LIN {X 0,Y 433.901,Z 245.879,A -85,B 0,C 180,E1 -10138.023,E2 -10138.023} C_VEL
LIN {X 0,Y 437.066,Z 265.172,A -85,B 0,C 180,E1 -10138.671,E2 -10138.671} C_VEL
LIN {X 0,Y 434.096,Z 394.919,A -85,B 0,C 180,E1 -10140.942,E2 -10140.942} C_VEL
LIN {X 0,Y 433.119,Z 438.839,A -85,B 0,C 180,E1 -10141.742,E2 -10141.742} C_VEL
LIN {X 0,Y 432.141,Z 454.828,A -85,B 0,C 180,E1 -10142.19,E2 -10142.19} C_VEL
LIN {X 0,Y 431.054,Z 471,A -85,B 0,C 180,E1 -10142.838,E2 -10142.838} C_VEL
LIN {X 0,Y 429.617,Z 486.877,A -85,B 0,C 180,E1 -10143.658,E2 -10143.658} C_VEL
LIN {X 0,Y 428.212,Z 501.806,A -85,B 0,C 180,E1 -10144.632,E2 -10144.632} C_VEL
LIN {X 0,Y 426.513,Z 516.607,A -85,B 0,C 180,E1 -10145.803,E2 -10145.803} C_VEL
LIN {X 0,Y 424.863,Z 530.394,A -85,B 0,C 180,E1 -10147.125,E2 -10147.125} C_VEL
LIN {X 0,Y 423.301,Z 543.183,A -85,B 0,C 180,E1 -10148.577,E2 -10148.577} C_VEL
LIN {X 0,Y 421.945,Z 554.232,A -85,B 0,C 180,E1 -10150.035,E2 -10150.035} C_VEL
LIN {X 0,Y 420.588,Z 565.241,A -85,B 0,C 180,E1 -10151.742,E2 -10151.742} C_VEL
LIN {X 0,Y 419.49,Z 575.91,A -85,B 0,C 180,E1 -10153.703,E2 -10153.703} C_VEL
LIN {X 0,Y 418.494,Z 584.872,A -85,B 0,C 180,E1 -10155.659,E2 -10155.659} C_VEL
LIN {X 0,Y 417.936,Z 591.553,A -85,B 0,C 180,E1 -10157.373,E2 -10157.373} C_VEL
LIN {X 0,Y 417.496,Z 597.846,A -85,B 0,C 180,E1 -10159.329,E2 -10159.329} C_VEL
LIN {X 0,Y 417.2,Z 603.006,A -85,B 0,C 180,E1 -10161.28,E2 -10161.28} C_VEL
LIN {X 0,Y 417.134,Z 607.023,A -85,B 0,C 180,E1 -10163.227,E2 -10163.227} C_VEL
LIN {X 0,Y 417.018,Z 609.993,A -85,B 0,C 180,E1 -10165.167,E2 -10165.167} C_VEL
LIN {X 0,Y 417.006,Z 611.955,A -85,B 0,C 180,E1 -10167.102,E2 -10167.102} C_VEL
LIN {X 0,Y 417.009,Z 612.924,A -85,B 0,C 180,E1 -10169.035,E2 -10169.035} C_VEL
LIN {X 0,Y 417.009,Z 612.93,A -85,B 0,C 180,E1 -10170.966,E2 -10170.966} C_VEL
LIN {X 0,Y 417.006,Z 611.951,A -85,B 0,C 180,E1 -10172.898,E2 -10172.898} C_VEL
LIN {X 0,Y 417.019,Z 609.997,A -85,B 0,C 180,E1 -10174.834,E2 -10174.834} C_VEL
LIN {X 0,Y 417.134,Z 607.013,A -85,B 0,C 180,E1 -10176.773,E2 -10176.773} C_VEL
LIN {X 0,Y 417.202,Z 602.998,A -85,B 0,C 180,E1 -10178.72,E2 -10178.72} C_VEL
LIN {X 0,Y 417.496,Z 597.807,A -85,B 0,C 180,E1 -10180.671,E2 -10180.671} C_VEL
LIN {X 0,Y 418.041,Z 590.748,A -85,B 0,C 180,E1 -10182.819,E2 -10182.819} C_VEL
LIN {X 0,Y 418.673,Z 582.701,A -85,B 0,C 180,E1 -10184.832,E2 -10184.832} C_VEL
LIN {X 0,Y 419.692,Z 573.308,A -85,B 0,C 180,E1 -10186.776,E2 -10186.776} C_VEL
LIN {X 0,Y 420.73,Z 563.461,A -85,B 0,C 180,E1 -10188.505,E2 -10188.505} C_VEL
LIN {X 0,Y 422.098,Z 552.064,A -85,B 0,C 180,E1 -10190.212,E2 -10190.212} C_VEL
LIN {X 0,Y 423.494,Z 540.698,A -85,B 0,C 180,E1 -10191.669,E2 -10191.669} C_VEL
LIN {X 0,Y 425.098,Z 527.299,A -85,B 0,C 180,E1 -10193.12,E2 -10193.12} C_VEL
LIN {X 0,Y 426.529,Z 514.146,A -85,B 0,C 180,E1 -10194.326,E2 -10194.326} C_VEL
LIN {X 0,Y 428.112,Z 499.325,A -85,B 0,C 180,E1 -10195.459,E2 -10195.459} C_VEL
LIN {X 0,Y 429.661,Z 484.109,A -85,B 0,C 180,E1 -10196.405,E2 -10196.405} C_VEL
LIN {X 0,Y 430.887,Z 468.48,A -85,B 0,C 180,E1 -10197.174,E2 -10197.174} C_VEL
LIN {X 0,Y 431.837,Z 452.772,A -85,B 0,C 180,E1 -10197.766,E2 -10197.766} C_VEL
LIN {X 0,Y 432.796,Z 435.249,A -85,B 0,C 180,E1 -10198.212,E2 -10198.212} C_VEL
LIN {X 0,Y 436.415,Z 265.637,A -85,B 0,C 180,E1 -10201.169,E2 -10201.169} C_VEL
LIN {X 0,Y 432.886,Z 244.933,A -85,B 0,C 180,E1 -10201.842,E2 -10201.842} C_VEL
LIN {X 0,Y 426.31,Z 230.903,A -85,B 0,C 180,E1 -10202.655,E2 -10202.655} C_VEL
LIN {X 0,Y 421.236,Z 214.637,A -85,B 0,C 180,E1 -10205.162,E2 -10205.162} C_VEL
LIN {X 0,Y 418.237,Z 205.705,A -85,B 0,C 180,E1 -10206.62,E2 -10206.62} C_VEL
LIN {X 0,Y 418.241,Z 205.695,A -85,B 0,C 180,E1 -10209.683,E2 -10209.683} C_VEL
LIN {X 0,Y 418.221,Z 205.698,A -85,B 0,C 180,E1 -10212.32,E2 -10212.32} C_VEL
LIN {X 0,Y 418.233,Z 205.696,A -85,B 0,C 180,E1 -10215.109,E2 -10215.109} C_VEL
LIN {X 0,Y 418.231,Z 205.701,A -85,B 0,C 180,E1 -10217.766,E2 -10217.766} C_VEL
LIN {X 0,Y 418.242,Z 205.7,A -85,B 0,C 180,E1 -10221.557,E2 -10221.557} C_VEL
LIN {X 0,Y 418.255,Z 205.699,A -85,B 0,C 180,E1 -10225.159,E2 -10225.159} C_VEL
LIN {X 0,Y 418.242,Z 205.69,A -85,B 0,C 180,E1 -10227.472,E2 -10227.472} C_VEL
LIN {X 0,Y 418.266,Z 205.7,A -85,B 0,C 180,E1 -10230.895,E2 -10230.895} C_VEL
LIN {X 0,Y 418.265,Z 205.679,A -85,B 0,C 180,E1 -10234.096,E2 -10234.096} C_VEL
LIN {X 0,Y 418.235,Z 205.7,A -85,B 0,C 180,E1 -10237.264,E2 -10237.264} C_VEL
LIN {X 0,Y 418.28,Z 205.676,A -85,B 0,C 180,E1 -10240.364,E2 -10240.364} C_VEL
LIN {X 0,Y 418.313,Z 205.687,A -85,B 0,C 180,E1 -10243.405,E2 -10243.405} C_VEL
LIN {X 0,Y 418.343,Z 205.669,A -85,B 0,C 180,E1 -10246.999,E2 -10246.999} C_VEL
LIN {X 0,Y 418.336,Z 205.676,A -85,B 0,C 180,E1 -10250.329,E2 -10250.329} C_VEL
LIN {X 0,Y 418.468,Z 205.668,A -85,B 0,C 180,E1 -10253.249,E2 -10253.249} C_VEL
LIN {X 0,Y 418.332,Z 205.673,A -85,B 0,C 180,E1 -10255.181,E2 -10255.181} C_VEL
LIN {X 0,Y 418.539,Z 205.636,A -85,B 0,C 180,E1 -10258.075,E2 -10258.075} C_VEL
LIN {X 0,Y 418.667,Z 205.639,A -85,B 0,C 180,E1 -10260,E2 -10260} C_VEL
LIN {X 0,Y 418.497,Z 205.662,A -85,B 0,C 180,E1 -10262.888,E2 -10262.888} C_VEL
LIN {X 0,Y 418.49,Z 205.664,A -85,B 0,C 180,E1 -10266.751,E2 -10266.751} C_VEL
LIN {X 0,Y 418.337,Z 205.686,A -85,B 0,C 180,E1 -10269.671,E2 -10269.671} C_VEL
LIN {X 0,Y 418.344,Z 205.675,A -85,B 0,C 180,E1 -10273.001,E2 -10273.001} C_VEL
LIN {X 0,Y 418.31,Z 205.684,A -85,B 0,C 180,E1 -10276.736,E2 -10276.736} C_VEL
LIN {X 0,Y 418.268,Z 205.683,A -85,B 0,C 180,E1 -10279.79,E2 -10279.79} C_VEL
LIN {X 0,Y 418.236,Z 205.696,A -85,B 0,C 180,E1 -10282.736,E2 -10282.736} C_VEL
LIN {X 0,Y 418.268,Z 205.683,A -85,B 0,C 180,E1 -10285.904,E2 -10285.904} C_VEL
LIN {X 0,Y 418.272,Z 205.694,A -85,B 0,C 180,E1 -10289.161,E2 -10289.161} C_VEL
LIN {X 0,Y 418.255,Z 205.686,A -85,B 0,C 180,E1 -10292.844,E2 -10292.844} C_VEL
LIN {X 0,Y 418.246,Z 205.694,A -85,B 0,C 180,E1 -10296.239,E2 -10296.239} C_VEL
LIN {X 0,Y 418.253,Z 205.695,A -85,B 0,C 180,E1 -10299.682,E2 -10299.682} C_VEL
LIN {X 0,Y 418.227,Z 205.696,A -85,B 0,C 180,E1 -10302.321,E2 -10302.321} C_VEL
LIN {X 0,Y 418.234,Z 205.694,A -85,B 0,C 180,E1 -10305.109,E2 -10305.109} C_VEL
LIN {X 0,Y 418.238,Z 205.695,A -85,B 0,C 180,E1 -10307.767,E2 -10307.767} C_VEL
LIN {X 0,Y 418.243,Z 205.695,A -85,B 0,C 180,E1 -10310.621,E2 -10310.621} C_VEL
LIN {X 0,Y 418.241,Z 205.689,A -85,B 0,C 180,E1 -10313.976,E2 -10313.976} C_VEL
LIN {X 0,Y 418.256,Z 205.699,A -85,B 0,C 180,E1 -10317.156,E2 -10317.156} C_VEL
LIN {X 0,Y 418.268,Z 205.698,A -85,B 0,C 180,E1 -10320.895,E2 -10320.895} C_VEL
LIN {X 0,Y 418.27,Z 205.694,A -85,B 0,C 180,E1 -10324.096,E2 -10324.096} C_VEL
LIN {X 0,Y 418.237,Z 205.699,A -85,B 0,C 180,E1 -10327.264,E2 -10327.264} C_VEL
LIN {X 0,Y 418.282,Z 205.675,A -85,B 0,C 180,E1 -10330.364,E2 -10330.364} C_VEL
LIN {X 0,Y 418.316,Z 205.695,A -85,B 0,C 180,E1 -10333.405,E2 -10333.405} C_VEL
LIN {X 0,Y 418.346,Z 205.672,A -85,B 0,C 180,E1 -10336.999,E2 -10336.999} C_VEL
LIN {X 0,Y 418.341,Z 205.689,A -85,B 0,C 180,E1 -10340.328,E2 -10340.328} C_VEL
LIN {X 0,Y 418.465,Z 205.835,A -85,B 0,C 180,E1 -10342.115,E2 -10342.115} C_VEL
LIN {X 0,Y 420.028,Z 210.56,A -85,B 0,C 180,E1 -10342.893,E2 -10342.893} C_VEL
LIN {X 0,Y 433.164,Z 236.683,A -85,B 0,C 180,E1 -10344.496,E2 -10344.496} C_VEL
LIN {X 0,Y 436.628,Z 244.26,A -85,B 0,C 180,E1 -10344.913,E2 -10344.913} C_VEL
LIN {X 0,Y 434.396,Z 345.325,A -85,B 0,C 180,E1 -10346.668,E2 -10346.668} C_VEL
LIN {X 0,Y 433.815,Z 351.169,A -85,B 0,C 180,E1 -10346.736,E2 -10346.736} C_VEL
LIN {X 0,Y 431.075,Z 360.699,A -85,B 0,C 180,E1 -10346.719,E2 -10346.719} C_VEL
LIN {X 0,Y 428.243,Z 370.233,A -85,B 0,C 180,E1 -10346.695,E2 -10346.695} C_VEL
LIN {X 0,Y 427.523,Z 376.09,A -85,B 0,C 180,E1 -10346.755,E2 -10346.755} C_VEL
LIN {X 0,Y 426.602,Z 416.506,A -85,B 0,C 180,E1 -10347.492,E2 -10347.492} C_VEL
LIN {X 0,Y 425.782,Z 433.559,A -85,B 0,C 180,E1 -10347.99,E2 -10347.99} C_VEL
LIN {X 0,Y 424.683,Z 449.382,A -85,B 0,C 180,E1 -10348.637,E2 -10348.637} C_VEL
LIN {X 0,Y 423.548,Z 463.898,A -85,B 0,C 180,E1 -10349.406,E2 -10349.406} C_VEL
LIN {X 0,Y 422.143,Z 478.979,A -85,B 0,C 180,E1 -10350.394,E2 -10350.394} C_VEL
LIN {X 0,Y 420.529,Z 493.459,A -85,B 0,C 180,E1 -10351.556,E2 -10351.556} C_VEL
LIN {X 0,Y 418.919,Z 507.193,A -85,B 0,C 180,E1 -10352.885,E2 -10352.885} C_VEL
LIN {X 0,Y 417.305,Z 519.957,A -85,B 0,C 180,E1 -10354.346,E2 -10354.346} C_VEL
LIN {X 0,Y 415.885,Z 530.987,A -85,B 0,C 180,E1 -10355.819,E2 -10355.819} C_VEL
LIN {X 0,Y 414.436,Z 541.968,A -85,B 0,C 180,E1 -10357.552,E2 -10357.552} C_VEL
LIN {X 0,Y 413.176,Z 551.925,A -85,B 0,C 180,E1 -10359.405,E2 -10359.405} C_VEL
LIN {X 0,Y 412.2,Z 560.572,A -85,B 0,C 180,E1 -10361.307,E2 -10361.307} C_VEL
LIN {X 0,Y 411.358,Z 568.645,A -85,B 0,C 180,E1 -10363.438,E2 -10363.438} C_VEL
LIN {X 0,Y 410.576,Z 576.071,A -85,B 0,C 180,E1 -10365.895,E2 -10365.895} C_VEL
LIN {X 0,Y 410.267,Z 580.899,A -85,B 0,C 180,E1 -10367.959,E2 -10367.959} C_VEL
LIN {X 0,Y 409.961,Z 584.63,A -85,B 0,C 180,E1 -10370.051,E2 -10370.051} C_VEL
LIN {X 0,Y 409.796,Z 587.298,A -85,B 0,C 180,E1 -10372.166,E2 -10372.166} C_VEL
LIN {X 0,Y 409.705,Z 588.922,A -85,B 0,C 180,E1 -10374.612,E2 -10374.612} C_VEL
LIN {X 0,Y 409.732,Z 589.098,A -85,B 0,C 180,E1 -10376.883,E2 -10376.883} C_VEL
LIN {X 0,Y 409.77,Z 588.172,A -85,B 0,C 180,E1 -10378.99,E2 -10378.99} C_VEL
LIN {X 0,Y 409.906,Z 586.261,A -85,B 0,C 180,E1 -10380.989,E2 -10380.989} C_VEL
LIN {X 0,Y 410.158,Z 582.863,A -85,B 0,C 180,E1 -10383.251,E2 -10383.251} C_VEL
LIN {X 0,Y 410.582,Z 577.94,A -85,B 0,C 180,E1 -10385.589,E2 -10385.589} C_VEL
LIN {X 0,Y 410.956,Z 573.155,A -85,B 0,C 180,E1 -10387.38,E2 -10387.38} C_VEL
LIN {X 0,Y 411.676,Z 566.16,A -85,B 0,C 180,E1 -10389.503,E2 -10389.503} C_VEL
LIN {X 0,Y 412.61,Z 557.646,A -85,B 0,C 180,E1 -10391.627,E2 -10391.627} C_VEL
LIN {X 0,Y 413.812,Z 548.585,A -85,B 0,C 180,E1 -10393.513,E2 -10393.513} C_VEL
LIN {X 0,Y 415.161,Z 538.348,A -85,B 0,C 180,E1 -10395.314,E2 -10395.314} C_VEL
LIN {X 0,Y 416.725,Z 526.906,A -85,B 0,C 180,E1 -10397.012,E2 -10397.012} C_VEL
LIN {X 0,Y 418.384,Z 514.662,A -85,B 0,C 180,E1 -10398.555,E2 -10398.555} C_VEL
LIN {X 0,Y 420.069,Z 501.652,A -85,B 0,C 180,E1 -10399.947,E2 -10399.947} C_VEL
LIN {X 0,Y 421.779,Z 487.222,A -85,B 0,C 180,E1 -10401.242,E2 -10401.242} C_VEL
LIN {X 0,Y 423.347,Z 472.399,A -85,B 0,C 180,E1 -10402.331,E2 -10402.331} C_VEL
LIN {X 0,Y 424.727,Z 457.148,A -85,B 0,C 180,E1 -10403.239,E2 -10403.239} C_VEL
LIN {X 0,Y 425.97,Z 440.485,A -85,B 0,C 180,E1 -10404.014,E2 -10404.014} C_VEL
LIN {X 0,Y 426.942,Z 423.926,A -85,B 0,C 180,E1 -10404.575,E2 -10404.575} C_VEL
LIN {X 0,Y 427.594,Z 406.333,A -85,B 0,C 180,E1 -10404.97,E2 -10404.97} C_VEL
LIN {X 0,Y 431.333,Z 247.058,A -85,B 0,C 180,E1 -10407.813,E2 -10407.813} C_VEL
LIN {X 0,Y 423.887,Z 231.742,A -85,B 0,C 180,E1 -10408.794,E2 -10408.794} C_VEL
LIN {X 0,Y 414.687,Z 214.868,A -85,B 0,C 180,E1 -10410.038,E2 -10410.038} C_VEL
LIN {X 0,Y 412.727,Z 211.295,A -85,B 0,C 180,E1 -10410.338,E2 -10410.338} C_VEL
LIN {X 0,Y 411.197,Z 206.576,A -85,B 0,C 180,E1 -10411.242,E2 -10411.242} C_VEL
LIN {X 0,Y 411.205,Z 206.573,A -85,B 0,C 180,E1 -10414.934,E2 -10414.934} C_VEL
LIN {X 0,Y 411.196,Z 206.57,A -85,B 0,C 180,E1 -10417.913,E2 -10417.913} C_VEL
LIN {X 0,Y 411.212,Z 206.57,A -85,B 0,C 180,E1 -10421.051,E2 -10421.051} C_VEL
LIN {X 0,Y 411.247,Z 206.563,A -85,B 0,C 180,E1 -10424.131,E2 -10424.131} C_VEL
LIN {X 0,Y 411.296,Z 206.558,A -85,B 0,C 180,E1 -10427.165,E2 -10427.165} C_VEL
LIN {X 0,Y 411.285,Z 206.567,A -85,B 0,C 180,E1 -10430.161,E2 -10430.161} C_VEL
LIN {X 0,Y 411.429,Z 206.545,A -85,B 0,C 180,E1 -10433.133,E2 -10433.133} C_VEL
LIN {X 0,Y 411.3,Z 206.561,A -85,B 0,C 180,E1 -10435.099,E2 -10435.099} C_VEL
LIN {X 0,Y 411.505,Z 206.537,A -85,B 0,C 180,E1 -10438.043,E2 -10438.043} C_VEL
LIN {X 0,Y 411.635,Z 206.523,A -85,B 0,C 180,E1 -10440,E2 -10440} C_VEL
LIN {X 0,Y 411.451,Z 206.54,A -85,B 0,C 180,E1 -10442.937,E2 -10442.937} C_VEL
LIN {X 0,Y 411.449,Z 206.545,A -85,B 0,C 180,E1 -10446.867,E2 -10446.867} C_VEL
LIN {X 0,Y 411.287,Z 206.568,A -85,B 0,C 180,E1 -10449.839,E2 -10449.839} C_VEL
LIN {X 0,Y 411.299,Z 206.562,A -85,B 0,C 180,E1 -10453.104,E2 -10453.104} C_VEL
LIN {X 0,Y 411.251,Z 206.566,A -85,B 0,C 180,E1 -10456.889,E2 -10456.889} C_VEL
LIN {X 0,Y 411.224,Z 206.576,A -85,B 0,C 180,E1 -10459.987,E2 -10459.987} C_VEL
LIN {X 0,Y 411.197,Z 206.577,A -85,B 0,C 180,E1 -10463.148,E2 -10463.148} C_VEL
LIN {X 0,Y 411.232,Z 206.568,A -85,B 0,C 180,E1 -10466.381,E2 -10466.381} C_VEL
LIN {X 0,Y 411.195,Z 206.579,A -85,B 0,C 180,E1 -10469.713,E2 -10469.713} C_VEL
LIN {X 0,Y 411.201,Z 206.58,A -85,B 0,C 180,E1 -10473.156,E2 -10473.156} C_VEL
LIN {X 0,Y 411.187,Z 206.58,A -85,B 0,C 180,E1 -10476.553,E2 -10476.553} C_VEL
LIN {X 0,Y 411.21,Z 206.579,A -85,B 0,C 180,E1 -10479.729,E2 -10479.729} C_VEL
LIN {X 0,Y 411.168,Z 206.589,A -85,B 0,C 180,E1 -10483.134,E2 -10483.134} C_VEL
LIN {X 0,Y 411.163,Z 206.585,A -85,B 0,C 180,E1 -10485.881,E2 -10485.881} C_VEL
LIN {X 0,Y 411.159,Z 206.584,A -85,B 0,C 180,E1 -10488.772,E2 -10488.772} C_VEL
LIN {X 0,Y 411.19,Z 206.578,A -85,B 0,C 180,E1 -10492.027,E2 -10492.027} C_VEL
LIN {X 0,Y 411.2,Z 206.646,A -85,B 0,C 180,E1 -10492.365,E2 -10492.365} C_VEL
LIN {X 0,Y 416.951,Z 223.259,A -85,B 0,C 180,E1 -10495.276,E2 -10495.276} C_VEL
LIN {X 0,Y 419.107,Z 230.043,A -85,B 0,C 180,E1 -10496.36,E2 -10496.36} C_VEL
LIN {X 0,Y 427.255,Z 246.676,A -85,B 0,C 180,E1 -10497.459,E2 -10497.459} C_VEL
LIN {X 0,Y 428.367,Z 249.681,A -85,B 0,C 180,E1 -10497.619,E2 -10497.619} C_VEL
LIN {X 0,Y 431.039,Z 266.077,A -85,B 0,C 180,E1 -10498.182,E2 -10498.182} C_VEL
LIN {X 0,Y 428.171,Z 385.084,A -85,B 0,C 180,E1 -10500.298,E2 -10500.298} C_VEL
LIN {X 0,Y 426.923,Z 438.456,A -85,B 0,C 180,E1 -10501.275,E2 -10501.275} C_VEL
LIN {X 0,Y 425.882,Z 454.998,A -85,B 0,C 180,E1 -10501.745,E2 -10501.745} C_VEL
LIN {X 0,Y 424.757,Z 471.045,A -85,B 0,C 180,E1 -10502.401,E2 -10502.401} C_VEL
LIN {X 0,Y 423.256,Z 486.837,A -85,B 0,C 180,E1 -10503.231,E2 -10503.231} C_VEL
LIN {X 0,Y 421.715,Z 501.754,A -85,B 0,C 180,E1 -10504.216,E2 -10504.216} C_VEL
LIN {X 0,Y 419.978,Z 516.482,A -85,B 0,C 180,E1 -10505.402,E2 -10505.402} C_VEL
LIN {X 0,Y 418.277,Z 530.255,A -85,B 0,C 180,E1 -10506.744,E2 -10506.744} C_VEL
LIN {X 0,Y 416.615,Z 543.032,A -85,B 0,C 180,E1 -10508.216,E2 -10508.216} C_VEL
LIN {X 0,Y 415.164,Z 554.071,A -85,B 0,C 180,E1 -10509.695,E2 -10509.695} C_VEL
LIN {X 0,Y 413.762,Z 565.079,A -85,B 0,C 180,E1 -10511.43,E2 -10511.43} C_VEL
LIN {X 0,Y 412.682,Z 574.487,A -85,B 0,C 180,E1 -10513.172,E2 -10513.172} C_VEL
LIN {X 0,Y 411.648,Z 583.662,A -85,B 0,C 180,E1 -10515.162,E2 -10515.162} C_VEL
LIN {X 0,Y 410.919,Z 591.36,A -85,B 0,C 180,E1 -10517.154,E2 -10517.154} C_VEL
LIN {X 0,Y 410.437,Z 597.652,A -85,B 0,C 180,E1 -10519.144,E2 -10519.144} C_VEL
LIN {X 0,Y 410.135,Z 602.81,A -85,B 0,C 180,E1 -10521.129,E2 -10521.129} C_VEL
LIN {X 0,Y 410.041,Z 606.827,A -85,B 0,C 180,E1 -10523.11,E2 -10523.11} C_VEL
LIN {X 0,Y 409.932,Z 609.794,A -85,B 0,C 180,E1 -10525.083,E2 -10525.083} C_VEL
LIN {X 0,Y 409.903,Z 611.755,A -85,B 0,C 180,E1 -10527.052,E2 -10527.052} C_VEL
LIN {X 0,Y 409.934,Z 612.721,A -85,B 0,C 180,E1 -10529.018,E2 -10529.018} C_VEL
LIN {X 0,Y 409.934,Z 612.724,A -85,B 0,C 180,E1 -10530.983,E2 -10530.983} C_VEL
LIN {X 0,Y 409.903,Z 611.738,A -85,B 0,C 180,E1 -10532.949,E2 -10532.949} C_VEL
LIN {X 0,Y 409.932,Z 609.781,A -85,B 0,C 180,E1 -10534.918,E2 -10534.918} C_VEL
LIN {X 0,Y 410.041,Z 606.79,A -85,B 0,C 180,E1 -10536.891,E2 -10536.891} C_VEL
LIN {X 0,Y 410.138,Z 602.771,A -85,B 0,C 180,E1 -10538.872,E2 -10538.872} C_VEL
LIN {X 0,Y 410.435,Z 597.569,A -85,B 0,C 180,E1 -10540.857,E2 -10540.857} C_VEL
LIN {X 0,Y 410.969,Z 591.016,A -85,B 0,C 180,E1 -10542.901,E2 -10542.901} C_VEL
LIN {X 0,Y 411.709,Z 582.442,A -85,B 0,C 180,E1 -10545.089,E2 -10545.089} C_VEL
LIN {X 0,Y 412.761,Z 573.118,A -85,B 0,C 180,E1 -10547.05,E2 -10547.05} C_VEL
LIN {X 0,Y 413.888,Z 563.179,A -85,B 0,C 180,E1 -10548.822,E2 -10548.822} C_VEL
LIN {X 0,Y 415.312,Z 551.759,A -85,B 0,C 180,E1 -10550.557,E2 -10550.557} C_VEL
LIN {X 0,Y 416.839,Z 539.807,A -85,B 0,C 180,E1 -10552.104,E2 -10552.104} C_VEL
LIN {X 0,Y 418.485,Z 526.935,A -85,B 0,C 180,E1 -10553.507,E2 -10553.507} C_VEL
LIN {X 0,Y 419.996,Z 513.732,A -85,B 0,C 180,E1 -10554.73,E2 -10554.73} C_VEL
LIN {X 0,Y 421.72,Z 498.303,A -85,B 0,C 180,E1 -10555.915,E2 -10555.915} C_VEL
LIN {X 0,Y 423.275,Z 483.583,A -85,B 0,C 180,E1 -10556.835,E2 -10556.835} C_VEL
LIN {X 0,Y 424.535,Z 467.894,A -85,B 0,C 180,E1 -10557.615,E2 -10557.615} C_VEL
LIN {X 0,Y 425.549,Z 452.033,A -85,B 0,C 180,E1 -10558.213,E2 -10558.213} C_VEL
LIN {X 0,Y 426.416,Z 436.159,A -85,B 0,C 180,E1 -10558.628,E2 -10558.628} C_VEL
LIN {X 0,Y 430.213,Z 265.8,A -85,B 0,C 180,E1 -10561.646,E2 -10561.646} C_VEL
LIN {X 0,Y 426.975,Z 247.562,A -85,B 0,C 180,E1 -10562.263,E2 -10562.263} C_VEL
LIN {X 0,Y 418.933,Z 230.448,A -85,B 0,C 180,E1 -10563.308,E2 -10563.308} C_VEL
LIN {X 0,Y 414.49,Z 216.465,A -85,B 0,C 180,E1 -10565.524,E2 -10565.524} C_VEL
LIN {X 0,Y 411.203,Z 206.575,A -85,B 0,C 180,E1 -10567.187,E2 -10567.187} C_VEL
LIN {X 0,Y 411.176,Z 206.575,A -85,B 0,C 180,E1 -10570.505,E2 -10570.505} C_VEL
LIN {X 0,Y 411.168,Z 206.576,A -85,B 0,C 180,E1 -10573.134,E2 -10573.134} C_VEL
LIN {X 0,Y 411.164,Z 206.572,A -85,B 0,C 180,E1 -10575.881,E2 -10575.881} C_VEL
LIN {X 0,Y 411.155,Z 206.577,A -85,B 0,C 180,E1 -10578.773,E2 -10578.773} C_VEL
LIN {X 0,Y 411.187,Z 206.578,A -85,B 0,C 180,E1 -10582.026,E2 -10582.026} C_VEL
LIN {X 0,Y 411.202,Z 206.575,A -85,B 0,C 180,E1 -10585.666,E2 -10585.666} C_VEL
LIN {X 0,Y 411.187,Z 206.569,A -85,B 0,C 180,E1 -10589.152,E2 -10589.152} C_VEL
LIN {X 0,Y 411.256,Z 206.564,A -85,B 0,C 180,E1 -10592.522,E2 -10592.522} C_VEL
LIN {X 0,Y 411.223,Z 206.568,A -85,B 0,C 180,E1 -10595.784,E2 -10595.784} C_VEL
LIN {X 0,Y 411.193,Z 206.568,A -85,B 0,C 180,E1 -10598.966,E2 -10598.966} C_VEL
LIN {X 0,Y 411.242,Z 206.557,A -85,B 0,C 180,E1 -10602.085,E2 -10602.085} C_VEL
LIN {X 0,Y 411.257,Z 206.566,A -85,B 0,C 180,E1 -10605.147,E2 -10605.147} C_VEL
LIN {X 0,Y 411.28,Z 206.542,A -85,B 0,C 180,E1 -10608.167,E2 -10608.167} C_VEL
LIN {X 0,Y 411.435,Z 206.547,A -85,B 0,C 180,E1 -10612.192,E2 -10612.192} C_VEL
LIN {X 0,Y 411.462,Z 206.54,A -85,B 0,C 180,E1 -10614.118,E2 -10614.118} C_VEL
LIN {X 0,Y 411.508,Z 206.511,A -85,B 0,C 180,E1 -10618.043,E2 -10618.043} C_VEL
LIN {X 0,Y 411.637,Z 206.515,A -85,B 0,C 180,E1 -10620,E2 -10620} C_VEL
LIN {X 0,Y 411.454,Z 206.539,A -85,B 0,C 180,E1 -10622.937,E2 -10622.937} C_VEL
LIN {X 0,Y 411.447,Z 206.537,A -85,B 0,C 180,E1 -10626.657,E2 -10626.657} C_VEL
LIN {X 0,Y 411.289,Z 206.564,A -85,B 0,C 180,E1 -10629.839,E2 -10629.839} C_VEL
LIN {X 0,Y 411.303,Z 206.552,A -85,B 0,C 180,E1 -10633.104,E2 -10633.104} C_VEL
LIN {X 0,Y 411.255,Z 206.562,A -85,B 0,C 180,E1 -10636.889,E2 -10636.889} C_VEL
LIN {X 0,Y 411.228,Z 206.562,A -85,B 0,C 180,E1 -10639.987,E2 -10639.987} C_VEL
LIN {X 0,Y 411.201,Z 206.573,A -85,B 0,C 180,E1 -10643.148,E2 -10643.148} C_VEL
LIN {X 0,Y 411.236,Z 206.564,A -85,B 0,C 180,E1 -10646.381,E2 -10646.381} C_VEL
LIN {X 0,Y 411.209,Z 206.576,A -85,B 0,C 180,E1 -10649.712,E2 -10649.712} C_VEL
LIN {X 0,Y 411.204,Z 206.565,A -85,B 0,C 180,E1 -10653.156,E2 -10653.156} C_VEL
LIN {X 0,Y 411.193,Z 206.571,A -85,B 0,C 180,E1 -10656.553,E2 -10656.553} C_VEL
LIN {X 0,Y 411.216,Z 206.572,A -85,B 0,C 180,E1 -10659.729,E2 -10659.729} C_VEL
LIN {X 0,Y 411.171,Z 206.574,A -85,B 0,C 180,E1 -10663.134,E2 -10663.134} C_VEL
LIN {X 0,Y 411.166,Z 206.582,A -85,B 0,C 180,E1 -10665.881,E2 -10665.881} C_VEL
LIN {X 0,Y 411.161,Z 206.573,A -85,B 0,C 180,E1 -10668.772,E2 -10668.772} C_VEL
LIN {X 0,Y 411.19,Z 206.575,A -85,B 0,C 180,E1 -10672.026,E2 -10672.026} C_VEL
LIN {X 0,Y 411.205,Z 206.578,A -85,B 0,C 180,E1 -10675.667,E2 -10675.667} C_VEL
LIN {X 0,Y 411.188,Z 206.571,A -85,B 0,C 180,E1 -10679.152,E2 -10679.152} C_VEL
LIN {X 0,Y 411.258,Z 206.563,A -85,B 0,C 180,E1 -10682.522,E2 -10682.522} C_VEL
LIN {X 0,Y 411.226,Z 206.566,A -85,B 0,C 180,E1 -10685.785,E2 -10685.785} C_VEL
LIN {X 0,Y 411.196,Z 206.573,A -85,B 0,C 180,E1 -10688.966,E2 -10688.966} C_VEL
LIN {X 0,Y 411.25,Z 206.556,A -85,B 0,C 180,E1 -10692.085,E2 -10692.085} C_VEL
LIN {X 0,Y 411.259,Z 206.556,A -85,B 0,C 180,E1 -10695.147,E2 -10695.147} C_VEL
LIN {X 0,Y 411.284,Z 206.567,A -85,B 0,C 180,E1 -10698.167,E2 -10698.167} C_VEL
LIN {X 0,Y 411.379,Z 206.592,A -85,B 0,C 180,E1 -10701.558,E2 -10701.558} C_VEL
LIN {X 0,Y 412.705,Z 210.66,A -85,B 0,C 180,E1 -10702.252,E2 -10702.252} C_VEL
LIN {X 0,Y 421.704,Z 228.197,A -85,B 0,C 180,E1 -10703.393,E2 -10703.393} C_VEL
LIN {X 0,Y 430.105,Z 245.542,A -85,B 0,C 180,E1 -10704.426,E2 -10704.426} C_VEL
LIN {X 0,Y 430.486,Z 246.607,A -85,B 0,C 180,E1 -10704.477,E2 -10704.477} C_VEL
LIN {X 0,Y 427.523,Z 376.09,A -85,B 0,C 180,E1 -10706.755,E2 -10706.755} C_VEL
LIN {X 0,Y 426.829,Z 381.941,A -85,B 0,C 180,E1 -10706.817,E2 -10706.817} C_VEL
LIN {X 0,Y 421.32,Z 401.012,A -85,B 0,C 180,E1 -10706.782,E2 -10706.782} C_VEL
LIN {X 0,Y 420.619,Z 406.863,A -85,B 0,C 180,E1 -10706.844,E2 -10706.844} C_VEL
LIN {X 0,Y 419.981,Z 424.149,A -85,B 0,C 180,E1 -10707.242,E2 -10707.242} C_VEL
LIN {X 0,Y 419.025,Z 440.472,A -85,B 0,C 180,E1 -10707.807,E2 -10707.807} C_VEL
LIN {X 0,Y 417.77,Z 456.503,A -85,B 0,C 180,E1 -10708.554,E2 -10708.554} C_VEL
LIN {X 0,Y 416.551,Z 470.709,A -85,B 0,C 180,E1 -10709.396,E2 -10709.396} C_VEL
LIN {X 0,Y 414.864,Z 486.123,A -85,B 0,C 180,E1 -10710.521,E2 -10710.521} C_VEL
LIN {X 0,Y 413.152,Z 500.721,A -85,B 0,C 180,E1 -10711.827,E2 -10711.827} C_VEL
LIN {X 0,Y 411.543,Z 513.411,A -85,B 0,C 180,E1 -10713.181,E2 -10713.181} C_VEL
LIN {X 0,Y 409.944,Z 525.353,A -85,B 0,C 180,E1 -10714.671,E2 -10714.671} C_VEL
LIN {X 0,Y 408.319,Z 537.248,A -85,B 0,C 180,E1 -10716.423,E2 -10716.423} C_VEL
LIN {X 0,Y 406.967,Z 547.339,A -85,B 0,C 180,E1 -10718.19,E2 -10718.19} C_VEL
LIN {X 0,Y 405.689,Z 557.197,A -85,B 0,C 180,E1 -10720.228,E2 -10720.228} C_VEL
LIN {X 0,Y 404.796,Z 564.575,A -85,B 0,C 180,E1 -10722.025,E2 -10722.025} C_VEL
LIN {X 0,Y 404.033,Z 571.607,A -85,B 0,C 180,E1 -10724.094,E2 -10724.094} C_VEL
LIN {X 0,Y 403.462,Z 577.388,A -85,B 0,C 180,E1 -10726.183,E2 -10726.183} C_VEL
LIN {X 0,Y 403.129,Z 582.034,A -85,B 0,C 180,E1 -10728.288,E2 -10728.288} C_VEL
LIN {X 0,Y 402.815,Z 585.508,A -85,B 0,C 180,E1 -10730.422,E2 -10730.422} C_VEL
LIN {X 0,Y 402.668,Z 587.884,A -85,B 0,C 180,E1 -10732.58,E2 -10732.58} C_VEL
LIN {X 0,Y 402.607,Z 589.212,A -85,B 0,C 180,E1 -10734.808,E2 -10734.808} C_VEL
LIN {X 0,Y 402.654,Z 589.274,A -85,B 0,C 180,E1 -10737.106,E2 -10737.106} C_VEL
LIN {X 0,Y 402.704,Z 588.221,A -85,B 0,C 180,E1 -10739.252,E2 -10739.252} C_VEL
LIN {X 0,Y 402.868,Z 585.901,A -85,B 0,C 180,E1 -10741.556,E2 -10741.556} C_VEL
LIN {X 0,Y 403.176,Z 582.165,A -85,B 0,C 180,E1 -10743.904,E2 -10743.904} C_VEL
LIN {X 0,Y 403.535,Z 578.333,A -85,B 0,C 180,E1 -10745.692,E2 -10745.692} C_VEL
LIN {X 0,Y 404.063,Z 572.1,A -85,B 0,C 180,E1 -10748.02,E2 -10748.02} C_VEL
LIN {X 0,Y 404.911,Z 564.75,A -85,B 0,C 180,E1 -10750.208,E2 -10750.208} C_VEL
LIN {X 0,Y 406.059,Z 555.468,A -85,B 0,C 180,E1 -10752.453,E2 -10752.453} C_VEL
LIN {X 0,Y 407.333,Z 546.13,A -85,B 0,C 180,E1 -10754.328,E2 -10754.328} C_VEL
LIN {X 0,Y 408.948,Z 535.094,A -85,B 0,C 180,E1 -10756.202,E2 -10756.202} C_VEL
LIN {X 0,Y 410.696,Z 522.725,A -85,B 0,C 180,E1 -10757.973,E2 -10757.973} C_VEL
LIN {X 0,Y 412.503,Z 509.604,A -85,B 0,C 180,E1 -10759.555,E2 -10759.555} C_VEL
LIN {X 0,Y 414.295,Z 496.239,A -85,B 0,C 180,E1 -10760.903,E2 -10760.903} C_VEL
LIN {X 0,Y 415.814,Z 483.264,A -85,B 0,C 180,E1 -10762.002,E2 -10762.002} C_VEL
LIN {X 0,Y 417.543,Z 467.508,A -85,B 0,C 180,E1 -10763.103,E2 -10763.103} C_VEL
LIN {X 0,Y 418.946,Z 451.699,A -85,B 0,C 180,E1 -10763.989,E2 -10763.989} C_VEL
LIN {X 0,Y 420.159,Z 435.395,A -85,B 0,C 180,E1 -10764.687,E2 -10764.687} C_VEL
LIN {X 0,Y 421.01,Z 419.267,A -85,B 0,C 180,E1 -10765.178,E2 -10765.178} C_VEL
LIN {X 0,Y 421.813,Z 390.17,A -85,B 0,C 180,E1 -10765.744,E2 -10765.744} C_VEL
LIN {X 0,Y 425.393,Z 249.294,A -85,B 0,C 180,E1 -10768.293,E2 -10768.293} C_VEL
LIN {X 0,Y 418.11,Z 234.407,A -85,B 0,C 180,E1 -10769.281,E2 -10769.281} C_VEL
LIN {X 0,Y 409.552,Z 218.725,A -85,B 0,C 180,E1 -10770.474,E2 -10770.474} C_VEL
LIN {X 0,Y 405.528,Z 211.614,A -85,B 0,C 180,E1 -10771.077,E2 -10771.077} C_VEL
LIN {X 0,Y 404.131,Z 207.46,A -85,B 0,C 180,E1 -10771.925,E2 -10771.925} C_VEL
LIN {X 0,Y 404.141,Z 207.451,A -85,B 0,C 180,E1 -10775.332,E2 -10775.332} C_VEL
LIN {X 0,Y 404.131,Z 207.454,A -85,B 0,C 180,E1 -10778.58,E2 -10778.58} C_VEL
LIN {X 0,Y 404.198,Z 207.448,A -85,B 0,C 180,E1 -10781.761,E2 -10781.761} C_VEL
LIN {X 0,Y 404.199,Z 207.442,A -85,B 0,C 180,E1 -10784.882,E2 -10784.882} C_VEL
LIN {X 0,Y 404.249,Z 207.431,A -85,B 0,C 180,E1 -10787.958,E2 -10787.958} C_VEL
LIN {X 0,Y 404.259,Z 207.439,A -85,B 0,C 180,E1 -10790.998,E2 -10790.998} C_VEL
LIN {X 0,Y 404.406,Z 207.421,A -85,B 0,C 180,E1 -10794.015,E2 -10794.015} C_VEL
LIN {X 0,Y 404.474,Z 207.413,A -85,B 0,C 180,E1 -10798.008,E2 -10798.008} C_VEL
LIN {X 0,Y 404.604,Z 207.399,A -85,B 0,C 180,E1 -10800,E2 -10800} C_VEL
LIN {X 0,Y 404.409,Z 207.417,A -85,B 0,C 180,E1 -10802.988,E2 -10802.988} C_VEL
LIN {X 0,Y 404.416,Z 207.42,A -85,B 0,C 180,E1 -10805.985,E2 -10805.985} C_VEL
LIN {X 0,Y 404.285,Z 207.436,A -85,B 0,C 180,E1 -10809.001,E2 -10809.001} C_VEL
LIN {X 0,Y 404.25,Z 207.443,A -85,B 0,C 180,E1 -10812.042,E2 -10812.042} C_VEL
LIN {X 0,Y 404.2,Z 207.447,A -85,B 0,C 180,E1 -10815.118,E2 -10815.118} C_VEL
LIN {X 0,Y 404.204,Z 207.446,A -85,B 0,C 180,E1 -10818.238,E2 -10818.238} C_VEL
LIN {X 0,Y 404.133,Z 207.456,A -85,B 0,C 180,E1 -10821.42,E2 -10821.42} C_VEL
LIN {X 0,Y 404.171,Z 207.449,A -85,B 0,C 180,E1 -10824.666,E2 -10824.666} C_VEL
LIN {X 0,Y 404.189,Z 207.451,A -85,B 0,C 180,E1 -10828,E2 -10828} C_VEL
LIN {X 0,Y 404.134,Z 207.457,A -85,B 0,C 180,E1 -10831.558,E2 -10831.558} C_VEL
LIN {X 0,Y 404.179,Z 207.456,A -85,B 0,C 180,E1 -10835.017,E2 -10835.017} C_VEL
LIN {X 0,Y 404.15,Z 207.459,A -85,B 0,C 180,E1 -10838.757,E2 -10838.757} C_VEL
LIN {X 0,Y 404.118,Z 207.463,A -85,B 0,C 180,E1 -10841.6,E2 -10841.6} C_VEL
LIN {X 0,Y 404.14,Z 207.461,A -85,B 0,C 180,E1 -10844.523,E2 -10844.523} C_VEL
LIN {X 0,Y 404.132,Z 207.461,A -85,B 0,C 180,E1 -10847.296,E2 -10847.296} C_VEL
LIN {X 0,Y 404.165,Z 207.455,A -85,B 0,C 180,E1 -10849.956,E2 -10849.956} C_VEL
LIN {X 0,Y 404.166,Z 207.528,A -85,B 0,C 180,E1 -10851.7,E2 -10851.7} C_VEL
LIN {X 0,Y 410.303,Z 225.065,A -85,B 0,C 180,E1 -10854.874,E2 -10854.874} C_VEL
LIN {X 0,Y 411.762,Z 229.615,A -85,B 0,C 180,E1 -10855.63,E2 -10855.63} C_VEL
LIN {X 0,Y 421.513,Z 249.283,A -85,B 0,C 180,E1 -10856.991,E2 -10856.991} C_VEL
LIN {X 0,Y 422.766,Z 252.707,A -85,B 0,C 180,E1 -10857.178,E2 -10857.178} C_VEL
LIN {X 0,Y 425.082,Z 267.338,A -85,B 0,C 180,E1 -10857.688,E2 -10857.688} C_VEL
LIN {X 0,Y 420.764,Z 438.216,A -85,B 0,C 180,E1 -10860.799,E2 -10860.799} C_VEL
LIN {X 0,Y 419.703,Z 454.259,A -85,B 0,C 180,E1 -10861.257,E2 -10861.257} C_VEL
LIN {X 0,Y 418.468,Z 471.099,A -85,B 0,C 180,E1 -10861.95,E2 -10861.95} C_VEL
LIN {X 0,Y 416.894,Z 486.826,A -85,B 0,C 180,E1 -10862.789,E2 -10862.789} C_VEL
LIN {X 0,Y 415.342,Z 501.122,A -85,B 0,C 180,E1 -10863.742,E2 -10863.742} C_VEL
LIN {X 0,Y 413.502,Z 516.408,A -85,B 0,C 180,E1 -10864.99,E2 -10864.99} C_VEL
LIN {X 0,Y 411.695,Z 530.139,A -85,B 0,C 180,E1 -10866.35,E2 -10866.35} C_VEL
LIN {X 0,Y 409.942,Z 542.885,A -85,B 0,C 180,E1 -10867.842,E2 -10867.842} C_VEL
LIN {X 0,Y 408.192,Z 555.554,A -85,B 0,C 180,E1 -10869.596,E2 -10869.596} C_VEL
LIN {X 0,Y 406.753,Z 566.366,A -85,B 0,C 180,E1 -10871.359,E2 -10871.359} C_VEL
LIN {X 0,Y 405.645,Z 575.564,A -85,B 0,C 180,E1 -10873.13,E2 -10873.13} C_VEL
LIN {X 0,Y 404.554,Z 584.507,A -85,B 0,C 180,E1 -10875.153,E2 -10875.153} C_VEL
LIN {X 0,Y 403.872,Z 591.526,A -85,B 0,C 180,E1 -10877.029,E2 -10877.029} C_VEL
LIN {X 0,Y 403.269,Z 598.901,A -85,B 0,C 180,E1 -10879.457,E2 -10879.457} C_VEL
LIN {X 0,Y 402.996,Z 604.787,A -85,B 0,C 180,E1 -10881.981,E2 -10881.981} C_VEL
LIN {X 0,Y 402.896,Z 608.23,A -85,B 0,C 180,E1 -10883.993,E2 -10883.993} C_VEL
LIN {X 0,Y 402.802,Z 610.73,A -85,B 0,C 180,E1 -10885.998,E2 -10885.998} C_VEL
LIN {X 0,Y 402.882,Z 612.146,A -85,B 0,C 180,E1 -10888.001,E2 -10888.001} C_VEL
LIN {X 0,Y 402.847,Z 612.671,A -85,B 0,C 180,E1 -10890,E2 -10890} C_VEL
LIN {X 0,Y 402.882,Z 612.133,A -85,B 0,C 180,E1 -10892,E2 -10892} C_VEL
LIN {X 0,Y 402.802,Z 610.7,A -85,B 0,C 180,E1 -10894.002,E2 -10894.002} C_VEL
LIN {X 0,Y 402.938,Z 607.929,A -85,B 0,C 180,E1 -10896.182,E2 -10896.182} C_VEL
LIN {X 0,Y 403.027,Z 603.624,A -85,B 0,C 180,E1 -10898.524,E2 -10898.524} C_VEL
LIN {X 0,Y 403.269,Z 598.773,A -85,B 0,C 180,E1 -10900.544,E2 -10900.544} C_VEL
LIN {X 0,Y 403.8,Z 592.786,A -85,B 0,C 180,E1 -10902.53,E2 -10902.53} C_VEL
LIN {X 0,Y 404.423,Z 585.274,A -85,B 0,C 180,E1 -10904.595,E2 -10904.595} C_VEL
LIN {X 0,Y 405.474,Z 576.435,A -85,B 0,C 180,E1 -10906.618,E2 -10906.618} C_VEL
LIN {X 0,Y 406.515,Z 567.279,A -85,B 0,C 180,E1 -10908.392,E2 -10908.392} C_VEL
LIN {X 0,Y 407.911,Z 556.557,A -85,B 0,C 180,E1 -10910.156,E2 -10910.156} C_VEL
LIN {X 0,Y 409.484,Z 544.699,A -85,B 0,C 180,E1 -10911.821,E2 -10911.821} C_VEL
LIN {X 0,Y 411.226,Z 531.291,A -85,B 0,C 180,E1 -10913.413,E2 -10913.413} C_VEL
LIN {X 0,Y 412.973,Z 517.589,A -85,B 0,C 180,E1 -10914.776,E2 -10914.776} C_VEL
LIN {X 0,Y 414.752,Z 502.403,A -85,B 0,C 180,E1 -10916.023,E2 -10916.023} C_VEL
LIN {X 0,Y 416.418,Z 487.224,A -85,B 0,C 180,E1 -10917.034,E2 -10917.034} C_VEL
LIN {X 0,Y 417.885,Z 471.214,A -85,B 0,C 180,E1 -10917.888,E2 -10917.888} C_VEL
LIN {X 0,Y 418.996,Z 454.947,A -85,B 0,C 180,E1 -10918.558,E2 -10918.558} C_VEL
LIN {X 0,Y 420.029,Z 438.436,A -85,B 0,C 180,E1 -10919.028,E2 -10919.028} C_VEL
LIN {X 0,Y 420.947,Z 400.568,A -85,B 0,C 180,E1 -10919.726,E2 -10919.726} C_VEL
LIN {X 0,Y 424.087,Z 266.896,A -85,B 0,C 180,E1 -10922.114,E2 -10922.114} C_VEL
LIN {X 0,Y 421.138,Z 250.26,A -85,B 0,C 180,E1 -10922.689,E2 -10922.689} C_VEL
LIN {X 0,Y 411.655,Z 230.281,A -85,B 0,C 180,E1 -10923.941,E2 -10923.941} C_VEL
LIN {X 0,Y 407.765,Z 218.253,A -85,B 0,C 180,E1 -10925.898,E2 -10925.898} C_VEL
LIN {X 0,Y 404.15,Z 207.452,A -85,B 0,C 180,E1 -10927.766,E2 -10927.766} C_VEL
LIN {X 0,Y 404.146,Z 207.45,A -85,B 0,C 180,E1 -10930.08,E2 -10930.08} C_VEL
LIN {X 0,Y 404.148,Z 207.45,A -85,B 0,C 180,E1 -10933.083,E2 -10933.083} C_VEL
LIN {X 0,Y 404.145,Z 207.446,A -85,B 0,C 180,E1 -10935.926,E2 -10935.926} C_VEL
LIN {X 0,Y 404.11,Z 207.456,A -85,B 0,C 180,E1 -10938.634,E2 -10938.634} C_VEL
LIN {X 0,Y 404.145,Z 207.457,A -85,B 0,C 180,E1 -10941.493,E2 -10941.493} C_VEL
LIN {X 0,Y 404.181,Z 207.448,A -85,B 0,C 180,E1 -10944.984,E2 -10944.984} C_VEL
LIN {X 0,Y 404.136,Z 207.442,A -85,B 0,C 180,E1 -10948.442,E2 -10948.442} C_VEL
LIN {X 0,Y 404.193,Z 207.448,A -85,B 0,C 180,E1 -10952,E2 -10952} C_VEL
LIN {X 0,Y 404.174,Z 207.445,A -85,B 0,C 180,E1 -10955.334,E2 -10955.334} C_VEL
LIN {X 0,Y 404.136,Z 207.452,A -85,B 0,C 180,E1 -10958.581,E2 -10958.581} C_VEL
LIN {X 0,Y 404.201,Z 207.432,A -85,B 0,C 180,E1 -10961.762,E2 -10961.762} C_VEL
LIN {X 0,Y 404.203,Z 207.447,A -85,B 0,C 180,E1 -10964.882,E2 -10964.882} C_VEL
LIN {X 0,Y 404.253,Z 207.417,A -85,B 0,C 180,E1 -10967.958,E2 -10967.958} C_VEL
LIN {X 0,Y 404.263,Z 207.438,A -85,B 0,C 180,E1 -10970.998,E2 -10970.998} C_VEL
LIN {X 0,Y 404.41,Z 207.42,A -85,B 0,C 180,E1 -10974.015,E2 -10974.015} C_VEL
LIN {X 0,Y 404.477,Z 207.385,A -85,B 0,C 180,E1 -10978.009,E2 -10978.009} C_VEL
LIN {X 0,Y 404.606,Z 207.39,A -85,B 0,C 180,E1 -10980,E2 -10980} C_VEL
LIN {X 0,Y 404.412,Z 207.416,A -85,B 0,C 180,E1 -10982.988,E2 -10982.988} C_VEL
LIN {X 0,Y 404.393,Z 207.414,A -85,B 0,C 180,E1 -10986.657,E2 -10986.657} C_VEL
LIN {X 0,Y 404.288,Z 207.434,A -85,B 0,C 180,E1 -10989.001,E2 -10989.001} C_VEL
LIN {X 0,Y 404.253,Z 207.426,A -85,B 0,C 180,E1 -10992.042,E2 -10992.042} C_VEL
LIN {X 0,Y 404.204,Z 207.444,A -85,B 0,C 180,E1 -10995.118,E2 -10995.118} C_VEL
LIN {X 0,Y 404.208,Z 207.43,A -85,B 0,C 180,E1 -10998.238,E2 -10998.238} C_VEL
LIN {X 0,Y 404.136,Z 207.453,A -85,B 0,C 180,E1 -11001.419,E2 -11001.419} C_VEL
LIN {X 0,Y 404.175,Z 207.438,A -85,B 0,C 180,E1 -11004.666,E2 -11004.666} C_VEL
LIN {X 0,Y 404.196,Z 207.451,A -85,B 0,C 180,E1 -11007.999,E2 -11007.999} C_VEL
LIN {X 0,Y 404.141,Z 207.444,A -85,B 0,C 180,E1 -11011.559,E2 -11011.559} C_VEL
LIN {X 0,Y 404.183,Z 207.449,A -85,B 0,C 180,E1 -11015.016,E2 -11015.016} C_VEL
LIN {X 0,Y 404.157,Z 207.441,A -85,B 0,C 180,E1 -11018.756,E2 -11018.756} C_VEL
LIN {X 0,Y 404.122,Z 207.459,A -85,B 0,C 180,E1 -11021.6,E2 -11021.6} C_VEL
LIN {X 0,Y 404.143,Z 207.446,A -85,B 0,C 180,E1 -11024.522,E2 -11024.522} C_VEL
LIN {X 0,Y 404.134,Z 207.458,A -85,B 0,C 180,E1 -11027.296,E2 -11027.296} C_VEL
LIN {X 0,Y 404.167,Z 207.45,A -85,B 0,C 180,E1 -11029.955,E2 -11029.955} C_VEL
LIN {X 0,Y 404.134,Z 207.451,A -85,B 0,C 180,E1 -11033.125,E2 -11033.125} C_VEL
LIN {X 0,Y 404.144,Z 207.455,A -85,B 0,C 180,E1 -11036.188,E2 -11036.188} C_VEL
LIN {X 0,Y 404.144,Z 207.455,A -85,B 0,C 180,E1 -11039.715,E2 -11039.715} C_VEL
LIN {X 0,Y 404.194,Z 207.443,A -85,B 0,C 180,E1 -11043.123,E2 -11043.123} C_VEL
LIN {X 0,Y 404.176,Z 207.449,A -85,B 0,C 180,E1 -11045.334,E2 -11045.334} C_VEL
LIN {X 0,Y 404.159,Z 207.455,A -85,B 0,C 180,E1 -11048.582,E2 -11048.582} C_VEL
LIN {X 0,Y 404.208,Z 207.428,A -85,B 0,C 180,E1 -11051.762,E2 -11051.762} C_VEL
LIN {X 0,Y 404.206,Z 207.438,A -85,B 0,C 180,E1 -11054.882,E2 -11054.882} C_VEL
LIN {X 0,Y 404.256,Z 207.442,A -85,B 0,C 180,E1 -11057.958,E2 -11057.958} C_VEL
LIN {X 0,Y 404.296,Z 207.488,A -85,B 0,C 180,E1 -11060.999,E2 -11060.999} C_VEL
LIN {X 0,Y 405.39,Z 210.828,A -85,B 0,C 180,E1 -11061.585,E2 -11061.585} C_VEL
LIN {X 0,Y 414.398,Z 227.936,A -85,B 0,C 180,E1 -11062.762,E2 -11062.762} C_VEL
LIN {X 0,Y 424.345,Z 248.403,A -85,B 0,C 180,E1 -11064.016,E2 -11064.016} C_VEL
LIN {X 0,Y 420.619,Z 406.863,A -85,B 0,C 180,E1 -11066.844,E2 -11066.844} C_VEL
LIN {X 0,Y 419.915,Z 412.704,A -85,B 0,C 180,E1 -11066.916,E2 -11066.916} C_VEL
LIN {X 0,Y 414.553,Z 429.706,A -85,B 0,C 180,E1 -11067.027,E2 -11067.027} C_VEL
LIN {X 0,Y 413.237,Z 435.408,A -85,B 0,C 180,E1 -11067.159,E2 -11067.159} C_VEL
LIN {X 0,Y 413.008,Z 437.279,A -85,B 0,C 180,E1 -11067.227,E2 -11067.227} C_VEL
LIN {X 0,Y 411.805,Z 453.028,A -85,B 0,C 180,E1 -11067.921,E2 -11067.921} C_VEL
LIN {X 0,Y 410.438,Z 467.836,A -85,B 0,C 180,E1 -11068.773,E2 -11068.773} C_VEL
LIN {X 0,Y 408.752,Z 483.365,A -85,B 0,C 180,E1 -11069.877,E2 -11069.877} C_VEL
LIN {X 0,Y 407.019,Z 497.628,A -85,B 0,C 180,E1 -11071.113,E2 -11071.113} C_VEL
LIN {X 0,Y 405.311,Z 510.878,A -85,B 0,C 180,E1 -11072.484,E2 -11072.484} C_VEL
LIN {X 0,Y 403.585,Z 523.14,A -85,B 0,C 180,E1 -11073.994,E2 -11073.994} C_VEL
LIN {X 0,Y 402.065,Z 533.812,A -85,B 0,C 180,E1 -11075.529,E2 -11075.529} C_VEL
LIN {X 0,Y 400.524,Z 544.453,A -85,B 0,C 180,E1 -11077.308,E2 -11077.308} C_VEL
LIN {X 0,Y 399.227,Z 553.6,A -85,B 0,C 180,E1 -11079.116,E2 -11079.116} C_VEL
LIN {X 0,Y 398.137,Z 562.463,A -85,B 0,C 180,E1 -11081.196,E2 -11081.196} C_VEL
LIN {X 0,Y 397.252,Z 570.046,A -85,B 0,C 180,E1 -11083.337,E2 -11083.337} C_VEL
LIN {X 0,Y 396.543,Z 576.118,A -85,B 0,C 180,E1 -11085.417,E2 -11085.417} C_VEL
LIN {X 0,Y 396.149,Z 581.009,A -85,B 0,C 180,E1 -11087.553,E2 -11087.553} C_VEL
LIN {X 0,Y 395.813,Z 584.909,A -85,B 0,C 180,E1 -11089.77,E2 -11089.77} C_VEL
LIN {X 0,Y 395.611,Z 587.554,A -85,B 0,C 180,E1 -11091.904,E2 -11091.904} C_VEL
LIN {X 0,Y 395.513,Z 589.112,A -85,B 0,C 180,E1 -11094.122,E2 -11094.122} C_VEL
LIN {X 0,Y 395.508,Z 589.592,A -85,B 0,C 180,E1 -11096.374,E2 -11096.374} C_VEL
LIN {X 0,Y 395.56,Z 588.885,A -85,B 0,C 180,E1 -11098.666,E2 -11098.666} C_VEL
LIN {X 0,Y 395.718,Z 586.88,A -85,B 0,C 180,E1 -11101,E2 -11101} C_VEL
LIN {X 0,Y 396.015,Z 583.372,A -85,B 0,C 180,E1 -11103.478,E2 -11103.478} C_VEL
LIN {X 0,Y 396.475,Z 578.729,A -85,B 0,C 180,E1 -11105.8,E2 -11105.8} C_VEL
LIN {X 0,Y 396.918,Z 573.964,A -85,B 0,C 180,E1 -11107.666,E2 -11107.666} C_VEL
LIN {X 0,Y 397.575,Z 568.269,A -85,B 0,C 180,E1 -11109.521,E2 -11109.521} C_VEL
LIN {X 0,Y 398.605,Z 560.102,A -85,B 0,C 180,E1 -11111.726,E2 -11111.726} C_VEL
LIN {X 0,Y 400.026,Z 550.184,A -85,B 0,C 180,E1 -11113.919,E2 -11113.919} C_VEL
LIN {X 0,Y 401.552,Z 539.683,A -85,B 0,C 180,E1 -11115.854,E2 -11115.854} C_VEL
LIN {X 0,Y 403.283,Z 528.463,A -85,B 0,C 180,E1 -11117.6,E2 -11117.6} C_VEL
LIN {X 0,Y 405.148,Z 515.873,A -85,B 0,C 180,E1 -11119.261,E2 -11119.261} C_VEL
LIN {X 0,Y 407.049,Z 502.737,A -85,B 0,C 180,E1 -11120.721,E2 -11120.721} C_VEL
LIN {X 0,Y 408.881,Z 488.387,A -85,B 0,C 180,E1 -11122.055,E2 -11122.055} C_VEL
LIN {X 0,Y 410.467,Z 474.992,A -85,B 0,C 180,E1 -11123.081,E2 -11123.081} C_VEL
LIN {X 0,Y 412.121,Z 458.81,A -85,B 0,C 180,E1 -11124.097,E2 -11124.097} C_VEL
LIN {X 0,Y 413.429,Z 442.652,A -85,B 0,C 180,E1 -11124.893,E2 -11124.893} C_VEL
LIN {X 0,Y 414.565,Z 425.998,A -85,B 0,C 180,E1 -11125.492,E2 -11125.492} C_VEL
LIN {X 0,Y 415.296,Z 408.925,A -85,B 0,C 180,E1 -11125.902,E2 -11125.902} C_VEL
LIN {X 0,Y 419.455,Z 252.075,A -85,B 0,C 180,E1 -11128.779,E2 -11128.779} C_VEL
LIN {X 0,Y 418.291,Z 249.071,A -85,B 0,C 180,E1 -11128.952,E2 -11128.952} C_VEL
LIN {X 0,Y 410.236,Z 233.005,A -85,B 0,C 180,E1 -11130.089,E2 -11130.089} C_VEL
LIN {X 0,Y 400.513,Z 215.767,A -85,B 0,C 180,E1 -11131.506,E2 -11131.506} C_VEL
LIN {X 0,Y 398.22,Z 211.897,A -85,B 0,C 180,E1 -11131.876,E2 -11131.876} C_VEL
LIN {X 0,Y 397.093,Z 208.332,A -85,B 0,C 180,E1 -11132.602,E2 -11132.602} C_VEL
LIN {X 0,Y 397.105,Z 208.331,A -85,B 0,C 180,E1 -11135.98,E2 -11135.98} C_VEL
LIN {X 0,Y 397.132,Z 208.331,A -85,B 0,C 180,E1 -11139.704,E2 -11139.704} C_VEL
LIN {X 0,Y 397.175,Z 208.326,A -85,B 0,C 180,E1 -11142.845,E2 -11142.845} C_VEL
LIN {X 0,Y 397.222,Z 208.316,A -85,B 0,C 180,E1 -11146.703,E2 -11146.703} C_VEL
LIN {X 0,Y 397.21,Z 208.318,A -85,B 0,C 180,E1 -11149.809,E2 -11149.809} C_VEL
LIN {X 0,Y 397.326,Z 208.303,A -85,B 0,C 180,E1 -11152.888,E2 -11152.888} C_VEL
LIN {X 0,Y 397.244,Z 208.314,A -85,B 0,C 180,E1 -11154.925,E2 -11154.925} C_VEL
LIN {X 0,Y 397.442,Z 208.289,A -85,B 0,C 180,E1 -11157.973,E2 -11157.973} C_VEL
LIN {X 0,Y 397.574,Z 208.275,A -85,B 0,C 180,E1 -11160,E2 -11160} C_VEL
LIN {X 0,Y 397.369,Z 208.294,A -85,B 0,C 180,E1 -11163.041,E2 -11163.041} C_VEL
LIN {X 0,Y 397.367,Z 208.298,A -85,B 0,C 180,E1 -11166.092,E2 -11166.092} C_VEL
LIN {X 0,Y 397.246,Z 208.312,A -85,B 0,C 180,E1 -11169.162,E2 -11169.162} C_VEL
LIN {X 0,Y 397.213,Z 208.321,A -85,B 0,C 180,E1 -11172.258,E2 -11172.258} C_VEL
LIN {X 0,Y 397.173,Z 208.324,A -85,B 0,C 180,E1 -11175.392,E2 -11175.392} C_VEL
LIN {X 0,Y 397.156,Z 208.322,A -85,B 0,C 180,E1 -11178.574,E2 -11178.574} C_VEL
LIN {X 0,Y 397.091,Z 208.332,A -85,B 0,C 180,E1 -11181.819,E2 -11181.819} C_VEL
LIN {X 0,Y 397.151,Z 208.325,A -85,B 0,C 180,E1 -11185.132,E2 -11185.132} C_VEL
LIN {X 0,Y 397.156,Z 208.329,A -85,B 0,C 180,E1 -11187.776,E2 -11187.776} C_VEL
LIN {X 0,Y 397.073,Z 208.338,A -85,B 0,C 180,E1 -11190.883,E2 -11190.883} C_VEL
LIN {X 0,Y 397.12,Z 208.333,A -85,B 0,C 180,E1 -11194.494,E2 -11194.494} C_VEL
LIN {X 0,Y 397.098,Z 208.336,A -85,B 0,C 180,E1 -11198.275,E2 -11198.275} C_VEL
LIN {X 0,Y 397.084,Z 208.341,A -85,B 0,C 180,E1 -11200.909,E2 -11200.909} C_VEL
LIN {X 0,Y 397.096,Z 208.338,A -85,B 0,C 180,E1 -11203.649,E2 -11203.649} C_VEL
LIN {X 0,Y 397.097,Z 208.34,A -85,B 0,C 180,E1 -11206.521,E2 -11206.521} C_VEL
LIN {X 0,Y 397.109,Z 208.332,A -85,B 0,C 180,E1 -11210.423,E2 -11210.423} C_VEL
LIN {X 0,Y 397.132,Z 208.466,A -85,B 0,C 180,E1 -11211.011,E2 -11211.011} C_VEL
LIN {X 0,Y 403.078,Z 225.31,A -85,B 0,C 180,E1 -11214.17,E2 -11214.17} C_VEL
LIN {X 0,Y 404.571,Z 229.602,A -85,B 0,C 180,E1 -11214.889,E2 -11214.889} C_VEL
LIN {X 0,Y 414.081,Z 248.436,A -85,B 0,C 180,E1 -11216.269,E2 -11216.269} C_VEL
LIN {X 0,Y 417.008,Z 254.779,A -85,B 0,C 180,E1 -11216.686,E2 -11216.686} C_VEL
LIN {X 0,Y 419.133,Z 268.817,A -85,B 0,C 180,E1 -11217.181,E2 -11217.181} C_VEL
LIN {X 0,Y 415.687,Z 396.969,A -85,B 0,C 180,E1 -11219.523,E2 -11219.523} C_VEL
LIN {X 0,Y 414.584,Z 438.757,A -85,B 0,C 180,E1 -11220.326,E2 -11220.326} C_VEL
LIN {X 0,Y 413.44,Z 455.376,A -85,B 0,C 180,E1 -11220.814,E2 -11220.814} C_VEL
LIN {X 0,Y 412.097,Z 472.449,A -85,B 0,C 180,E1 -11221.547,E2 -11221.547} C_VEL
LIN {X 0,Y 410.568,Z 486.816,A -85,B 0,C 180,E1 -11222.335,E2 -11222.335} C_VEL
LIN {X 0,Y 408.845,Z 501.899,A -85,B 0,C 180,E1 -11223.364,E2 -11223.364} C_VEL
LIN {X 0,Y 407.009,Z 516.336,A -85,B 0,C 180,E1 -11224.563,E2 -11224.563} C_VEL
LIN {X 0,Y 405.132,Z 530.047,A -85,B 0,C 180,E1 -11225.942,E2 -11225.942} C_VEL
LIN {X 0,Y 403.261,Z 542.874,A -85,B 0,C 180,E1 -11227.469,E2 -11227.469} C_VEL
LIN {X 0,Y 401.446,Z 555.414,A -85,B 0,C 180,E1 -11229.237,E2 -11229.237} C_VEL
LIN {X 0,Y 399.917,Z 566.202,A -85,B 0,C 180,E1 -11231.028,E2 -11231.028} C_VEL
LIN {X 0,Y 398.613,Z 576.643,A -85,B 0,C 180,E1 -11233.088,E2 -11233.088} C_VEL
LIN {X 0,Y 397.466,Z 585.355,A -85,B 0,C 180,E1 -11235.145,E2 -11235.145} C_VEL
LIN {X 0,Y 396.733,Z 593.037,A -85,B 0,C 180,E1 -11237.329,E2 -11237.329} C_VEL
LIN {X 0,Y 396.226,Z 598.718,A -85,B 0,C 180,E1 -11239.267,E2 -11239.267} C_VEL
LIN {X 0,Y 395.911,Z 604.599,A -85,B 0,C 180,E1 -11241.836,E2 -11241.836} C_VEL
LIN {X 0,Y 395.819,Z 608.035,A -85,B 0,C 180,E1 -11243.885,E2 -11243.885} C_VEL
LIN {X 0,Y 395.724,Z 610.531,A -85,B 0,C 180,E1 -11245.927,E2 -11245.927} C_VEL
LIN {X 0,Y 395.778,Z 611.944,A -85,B 0,C 180,E1 -11247.965,E2 -11247.965} C_VEL
LIN {X 0,Y 395.774,Z 612.465,A -85,B 0,C 180,E1 -11250,E2 -11250} C_VEL
LIN {X 0,Y 395.779,Z 611.924,A -85,B 0,C 180,E1 -11252.036,E2 -11252.036} C_VEL
LIN {X 0,Y 395.725,Z 610.485,A -85,B 0,C 180,E1 -11254.074,E2 -11254.074} C_VEL
LIN {X 0,Y 395.819,Z 607.965,A -85,B 0,C 180,E1 -11256.116,E2 -11256.116} C_VEL
LIN {X 0,Y 395.912,Z 604.475,A -85,B 0,C 180,E1 -11258.164,E2 -11258.164} C_VEL
LIN {X 0,Y 396.088,Z 599.834,A -85,B 0,C 180,E1 -11260.221,E2 -11260.221} C_VEL
LIN {X 0,Y 396.632,Z 594.052,A -85,B 0,C 180,E1 -11262.277,E2 -11262.277} C_VEL
LIN {X 0,Y 397.247,Z 587.035,A -85,B 0,C 180,E1 -11264.341,E2 -11264.341} C_VEL
LIN {X 0,Y 398.421,Z 577.373,A -85,B 0,C 180,E1 -11266.657,E2 -11266.657} C_VEL
LIN {X 0,Y 399.636,Z 566.976,A -85,B 0,C 180,E1 -11268.72,E2 -11268.72} C_VEL
LIN {X 0,Y 401.127,Z 556.234,A -85,B 0,C 180,E1 -11270.513,E2 -11270.513} C_VEL
LIN {X 0,Y 402.874,Z 543.821,A -85,B 0,C 180,E1 -11272.271,E2 -11272.271} C_VEL
LIN {X 0,Y 404.467,Z 532.096,A -85,B 0,C 180,E1 -11273.692,E2 -11273.692} C_VEL
LIN {X 0,Y 406.273,Z 518.497,A -85,B 0,C 180,E1 -11275.076,E2 -11275.076} C_VEL
LIN {X 0,Y 408.074,Z 504.1,A -85,B 0,C 180,E1 -11276.297,E2 -11276.297} C_VEL
LIN {X 0,Y 409.732,Z 489.619,A -85,B 0,C 180,E1 -11277.312,E2 -11277.312} C_VEL
LIN {X 0,Y 411.28,Z 474.523,A -85,B 0,C 180,E1 -11278.168,E2 -11278.168} C_VEL
LIN {X 0,Y 412.583,Z 456.882,A -85,B 0,C 180,E1 -11278.939,E2 -11278.939} C_VEL
LIN {X 0,Y 413.682,Z 439.838,A -85,B 0,C 180,E1 -11279.447,E2 -11279.447} C_VEL
LIN {X 0,Y 414.485,Z 413.669,A -85,B 0,C 180,E1 -11279.951,E2 -11279.951} C_VEL
LIN {X 0,Y 418.012,Z 268.951,A -85,B 0,C 180,E1 -11282.572,E2 -11282.572} C_VEL
LIN {X 0,Y 415.653,Z 253.74,A -85,B 0,C 180,E1 -11283.081,E2 -11283.081} C_VEL
LIN {X 0,Y 405.717,Z 233.047,A -85,B 0,C 180,E1 -11284.392,E2 -11284.392} C_VEL
LIN {X 0,Y 404.392,Z 230.238,A -85,B 0,C 180,E1 -11284.58,E2 -11284.58} C_VEL
LIN {X 0,Y 399.43,Z 215.194,A -85,B 0,C 180,E1 -11287.119,E2 -11287.119} C_VEL
LIN {X 0,Y 397.102,Z 208.334,A -85,B 0,C 180,E1 -11288.348,E2 -11288.348} C_VEL
LIN {X 0,Y 397.085,Z 208.334,A -85,B 0,C 180,E1 -11290.909,E2 -11290.909} C_VEL
LIN {X 0,Y 397.098,Z 208.333,A -85,B 0,C 180,E1 -11293.649,E2 -11293.649} C_VEL
LIN {X 0,Y 397.098,Z 208.327,A -85,B 0,C 180,E1 -11296.521,E2 -11296.521} C_VEL
LIN {X 0,Y 397.088,Z 208.33,A -85,B 0,C 180,E1 -11300.42,E2 -11300.42} C_VEL
LIN {X 0,Y 397.095,Z 208.323,A -85,B 0,C 180,E1 -11303.005,E2 -11303.005} C_VEL
LIN {X 0,Y 397.116,Z 208.331,A -85,B 0,C 180,E1 -11306.282,E2 -11306.282} C_VEL
LIN {X 0,Y 397.102,Z 208.328,A -85,B 0,C 180,E1 -11310.135,E2 -11310.135} C_VEL
LIN {X 0,Y 397.192,Z 208.314,A -85,B 0,C 180,E1 -11312.61,E2 -11312.61} C_VEL
LIN {X 0,Y 397.13,Z 208.324,A -85,B 0,C 180,E1 -11315.982,E2 -11315.982} C_VEL
LIN {X 0,Y 397.136,Z 208.315,A -85,B 0,C 180,E1 -11319.705,E2 -11319.705} C_VEL
LIN {X 0,Y 397.179,Z 208.318,A -85,B 0,C 180,E1 -11322.845,E2 -11322.845} C_VEL
LIN {X 0,Y 397.226,Z 208.301,A -85,B 0,C 180,E1 -11326.703,E2 -11326.703} C_VEL
LIN {X 0,Y 397.214,Z 208.301,A -85,B 0,C 180,E1 -11329.809,E2 -11329.809} C_VEL
LIN {X 0,Y 397.33,Z 208.303,A -85,B 0,C 180,E1 -11332.888,E2 -11332.888} C_VEL
LIN {X 0,Y 397.247,Z 208.3,A -85,B 0,C 180,E1 -11334.925,E2 -11334.925} C_VEL
LIN {X 0,Y 397.446,Z 208.26,A -85,B 0,C 180,E1 -11337.973,E2 -11337.973} C_VEL
LIN {X 0,Y 397.576,Z 208.266,A -85,B 0,C 180,E1 -11340,E2 -11340} C_VEL
LIN {X 0,Y 397.372,Z 208.293,A -85,B 0,C 180,E1 -11343.041,E2 -11343.041} C_VEL
LIN {X 0,Y 397.344,Z 208.291,A -85,B 0,C 180,E1 -11346.655,E2 -11346.655} C_VEL
LIN {X 0,Y 397.25,Z 208.311,A -85,B 0,C 180,E1 -11349.162,E2 -11349.162} C_VEL
LIN {X 0,Y 397.216,Z 208.303,A -85,B 0,C 180,E1 -11352.258,E2 -11352.258} C_VEL
LIN {X 0,Y 397.177,Z 208.321,A -85,B 0,C 180,E1 -11355.392,E2 -11355.392} C_VEL
LIN {X 0,Y 397.16,Z 208.306,A -85,B 0,C 180,E1 -11358.573,E2 -11358.573} C_VEL
LIN {X 0,Y 397.094,Z 208.334,A -85,B 0,C 180,E1 -11361.819,E2 -11361.819} C_VEL
LIN {X 0,Y 397.154,Z 208.311,A -85,B 0,C 180,E1 -11365.132,E2 -11365.132} C_VEL
LIN {X 0,Y 397.161,Z 208.323,A -85,B 0,C 180,E1 -11367.777,E2 -11367.777} C_VEL
LIN {X 0,Y 397.082,Z 208.327,A -85,B 0,C 180,E1 -11370.882,E2 -11370.882} C_VEL
LIN {X 0,Y 397.124,Z 208.328,A -85,B 0,C 180,E1 -11374.493,E2 -11374.493} C_VEL
LIN {X 0,Y 397.105,Z 208.319,A -85,B 0,C 180,E1 -11378.275,E2 -11378.275} C_VEL
LIN {X 0,Y 397.088,Z 208.333,A -85,B 0,C 180,E1 -11380.909,E2 -11380.909} C_VEL
LIN {X 0,Y 397.099,Z 208.322,A -85,B 0,C 180,E1 -11383.649,E2 -11383.649} C_VEL
LIN {X 0,Y 397.1,Z 208.331,A -85,B 0,C 180,E1 -11386.521,E2 -11386.521} C_VEL
LIN {X 0,Y 397.111,Z 208.328,A -85,B 0,C 180,E1 -11390.423,E2 -11390.423} C_VEL
LIN {X 0,Y 397.107,Z 208.321,A -85,B 0,C 180,E1 -11394.265,E2 -11394.265} C_VEL
LIN {X 0,Y 397.114,Z 208.332,A -85,B 0,C 180,E1 -11396.727,E2 -11396.727} C_VEL
LIN {X 0,Y 397.123,Z 208.329,A -85,B 0,C 180,E1 -11400.296,E2 -11400.296} C_VEL
LIN {X 0,Y 397.193,Z 208.314,A -85,B 0,C 180,E1 -11402.61,E2 -11402.61} C_VEL
LIN {X 0,Y 397.132,Z 208.321,A -85,B 0,C 180,E1 -11405.982,E2 -11405.982} C_VEL
LIN {X 0,Y 397.138,Z 208.315,A -85,B 0,C 180,E1 -11409.705,E2 -11409.705} C_VEL
LIN {X 0,Y 397.181,Z 208.319,A -85,B 0,C 180,E1 -11412.845,E2 -11412.845} C_VEL
LIN {X 0,Y 397.228,Z 208.297,A -85,B 0,C 180,E1 -11416.703,E2 -11416.703} C_VEL
LIN {X 0,Y 397.239,Z 208.372,A -85,B 0,C 180,E1 -11420.42,E2 -11420.42} C_VEL
LIN {X 0,Y 398.244,Z 211.246,A -85,B 0,C 180,E1 -11420.917,E2 -11420.917} C_VEL
LIN {X 0,Y 407.355,Z 228.277,A -85,B 0,C 180,E1 -11422.14,E2 -11422.14} C_VEL
LIN {X 0,Y 418.134,Z 250.279,A -85,B 0,C 180,E1 -11423.541,E2 -11423.541} C_VEL
LIN {X 0,Y 414.834,Z 387.129,A -85,B 0,C 180,E1 -11426.023,E2 -11426.023} C_VEL
LIN {X 0,Y 413.993,Z 418.301,A -85,B 0,C 180,E1 -11426.624,E2 -11426.624} C_VEL
LIN {X 0,Y 413.13,Z 435.012,A -85,B 0,C 180,E1 -11427.135,E2 -11427.135} C_VEL
LIN {X 0,Y 413.008,Z 437.279,A -85,B 0,C 180,E1 -11427.227,E2 -11427.227} C_VEL
LIN {X 0,Y 412.369,Z 441.06,A -85,B 0,C 180,E1 -11427.35,E2 -11427.35} C_VEL
LIN {X 0,Y 408.561,Z 452.132,A -85,B 0,C 180,E1 -11427.638,E2 -11427.638} C_VEL
LIN {X 0,Y 405.296,Z 461.236,A -85,B 0,C 180,E1 -11427.952,E2 -11427.952} C_VEL
LIN {X 0,Y 404.196,Z 466.597,A -85,B 0,C 180,E1 -11428.242,E2 -11428.242} C_VEL
LIN {X 0,Y 402.412,Z 482.6,A -85,B 0,C 180,E1 -11429.374,E2 -11429.374} C_VEL
LIN {X 0,Y 400.618,Z 496.933,A -85,B 0,C 180,E1 -11430.616,E2 -11430.616} C_VEL
LIN {X 0,Y 398.791,Z 510.436,A -85,B 0,C 180,E1 -11432.02,E2 -11432.02} C_VEL
LIN {X 0,Y 397.012,Z 522.775,A -85,B 0,C 180,E1 -11433.552,E2 -11433.552} C_VEL
LIN {X 0,Y 395.243,Z 534.607,A -85,B 0,C 180,E1 -11435.279,E2 -11435.279} C_VEL
LIN {X 0,Y 393.574,Z 545.632,A -85,B 0,C 180,E1 -11437.18,E2 -11437.18} C_VEL
LIN {X 0,Y 392.237,Z 554.699,A -85,B 0,C 180,E1 -11439.02,E2 -11439.02} C_VEL
LIN {X 0,Y 391.092,Z 563.41,A -85,B 0,C 180,E1 -11441.138,E2 -11441.138} C_VEL
LIN {X 0,Y 390.141,Z 571.119,A -85,B 0,C 180,E1 -11443.406,E2 -11443.406} C_VEL
LIN {X 0,Y 389.417,Z 577.436,A -85,B 0,C 180,E1 -11445.706,E2 -11445.706} C_VEL
LIN {X 0,Y 389.038,Z 582.167,A -85,B 0,C 180,E1 -11447.884,E2 -11447.884} C_VEL
LIN {X 0,Y 388.67,Z 585.7,A -85,B 0,C 180,E1 -11450.093,E2 -11450.093} C_VEL
LIN {X 0,Y 388.481,Z 588.449,A -85,B 0,C 180,E1 -11452.685,E2 -11452.685} C_VEL
LIN {X 0,Y 388.413,Z 589.691,A -85,B 0,C 180,E1 -11455.216,E2 -11455.216} C_VEL
LIN {X 0,Y 388.475,Z 589.609,A -85,B 0,C 180,E1 -11457.567,E2 -11457.567} C_VEL
LIN {X 0,Y 388.541,Z 588.37,A -85,B 0,C 180,E1 -11459.746,E2 -11459.746} C_VEL
LIN {X 0,Y 388.721,Z 586.273,A -85,B 0,C 180,E1 -11461.816,E2 -11461.816} C_VEL
LIN {X 0,Y 389.067,Z 582.857,A -85,B 0,C 180,E1 -11464.053,E2 -11464.053} C_VEL
LIN {X 0,Y 389.375,Z 579.648,A -85,B 0,C 180,E1 -11465.687,E2 -11465.687} C_VEL
LIN {X 0,Y 389.881,Z 574.425,A -85,B 0,C 180,E1 -11467.797,E2 -11467.797} C_VEL
LIN {X 0,Y 390.613,Z 568.521,A -85,B 0,C 180,E1 -11469.767,E2 -11469.767} C_VEL
LIN {X 0,Y 391.634,Z 560.825,A -85,B 0,C 180,E1 -11471.894,E2 -11471.894} C_VEL
LIN {X 0,Y 392.934,Z 552.187,A -85,B 0,C 180,E1 -11473.873,E2 -11473.873} C_VEL
LIN {X 0,Y 394.42,Z 542.572,A -85,B 0,C 180,E1 -11475.75,E2 -11475.75} C_VEL
LIN {X 0,Y 396.285,Z 531.164,A -85,B 0,C 180,E1 -11477.63,E2 -11477.63} C_VEL
LIN {X 0,Y 398.246,Z 518.691,A -85,B 0,C 180,E1 -11479.36,E2 -11479.36} C_VEL
LIN {X 0,Y 400.239,Z 505.326,A -85,B 0,C 180,E1 -11480.91,E2 -11480.91} C_VEL
LIN {X 0,Y 402.231,Z 490.993,A -85,B 0,C 180,E1 -11482.299,E2 -11482.299} C_VEL
LIN {X 0,Y 404.017,Z 476.856,A -85,B 0,C 180,E1 -11483.436,E2 -11483.436} C_VEL
LIN {X 0,Y 405.598,Z 462.518,A -85,B 0,C 180,E1 -11484.389,E2 -11484.389} C_VEL
LIN {X 0,Y 407.099,Z 445.651,A -85,B 0,C 180,E1 -11485.271,E2 -11485.271} C_VEL
LIN {X 0,Y 408.317,Z 428.986,A -85,B 0,C 180,E1 -11485.907,E2 -11485.907} C_VEL
LIN {X 0,Y 409.116,Z 412.323,A -85,B 0,C 180,E1 -11486.344,E2 -11486.344} C_VEL
LIN {X 0,Y 413.515,Z 253.744,A -85,B 0,C 180,E1 -11489.311,E2 -11489.311} C_VEL
LIN {X 0,Y 405.557,Z 237.667,A -85,B 0,C 180,E1 -11490.464,E2 -11490.464} C_VEL
LIN {X 0,Y 396.178,Z 220.771,A -85,B 0,C 180,E1 -11491.873,E2 -11491.873} C_VEL
LIN {X 0,Y 391.097,Z 212.204,A -85,B 0,C 180,E1 -11492.691,E2 -11492.691} C_VEL
LIN {X 0,Y 390.031,Z 209.21,A -85,B 0,C 180,E1 -11493.345,E2 -11493.345} C_VEL
LIN {X 0,Y 390.058,Z 209.213,A -85,B 0,C 180,E1 -11496.765,E2 -11496.765} C_VEL
LIN {X 0,Y 390.097,Z 209.206,A -85,B 0,C 180,E1 -11499.983,E2 -11499.983} C_VEL
LIN {X 0,Y 390.131,Z 209.199,A -85,B 0,C 180,E1 -11503.248,E2 -11503.248} C_VEL
LIN {X 0,Y 390.188,Z 209.194,A -85,B 0,C 180,E1 -11506.561,E2 -11506.561} C_VEL
LIN {X 0,Y 390.161,Z 209.196,A -85,B 0,C 180,E1 -11509.623,E2 -11509.623} C_VEL
LIN {X 0,Y 390.274,Z 209.182,A -85,B 0,C 180,E1 -11512.758,E2 -11512.758} C_VEL
LIN {X 0,Y 390.215,Z 209.19,A -85,B 0,C 180,E1 -11514.833,E2 -11514.833} C_VEL
LIN {X 0,Y 390.411,Z 209.164,A -85,B 0,C 180,E1 -11517.937,E2 -11517.937} C_VEL
LIN {X 0,Y 390.543,Z 209.15,A -85,B 0,C 180,E1 -11520,E2 -11520} C_VEL
LIN {X 0,Y 390.304,Z 209.174,A -85,B 0,C 180,E1 -11523.097,E2 -11523.097} C_VEL
LIN {X 0,Y 390.321,Z 209.176,A -85,B 0,C 180,E1 -11526.202,E2 -11526.202} C_VEL
LIN {X 0,Y 390.199,Z 209.191,A -85,B 0,C 180,E1 -11529.329,E2 -11529.329} C_VEL
LIN {X 0,Y 390.188,Z 209.192,A -85,B 0,C 180,E1 -11533.439,E2 -11533.439} C_VEL
LIN {X 0,Y 390.142,Z 209.197,A -85,B 0,C 180,E1 -11537.308,E2 -11537.308} C_VEL
LIN {X 0,Y 390.081,Z 209.207,A -85,B 0,C 180,E1 -11540.47,E2 -11540.47} C_VEL
LIN {X 0,Y 390.084,Z 209.209,A -85,B 0,C 180,E1 -11543.351,E2 -11543.351} C_VEL
LIN {X 0,Y 390.108,Z 209.199,A -85,B 0,C 180,E1 -11546.768,E2 -11546.768} C_VEL
LIN {X 0,Y 390.033,Z 209.214,A -85,B 0,C 180,E1 -11550.3,E2 -11550.3} C_VEL
LIN {X 0,Y 390.063,Z 209.211,A -85,B 0,C 180,E1 -11554.025,E2 -11554.025} C_VEL
LIN {X 0,Y 390.038,Z 209.217,A -85,B 0,C 180,E1 -11557.551,E2 -11557.551} C_VEL
LIN {X 0,Y 390.051,Z 209.217,A -85,B 0,C 180,E1 -11560.822,E2 -11560.822} C_VEL
LIN {X 0,Y 390.05,Z 209.215,A -85,B 0,C 180,E1 -11563.887,E2 -11563.887} C_VEL
LIN {X 0,Y 390.053,Z 209.217,A -85,B 0,C 180,E1 -11566.79,E2 -11566.79} C_VEL
LIN {X 0,Y 390.072,Z 209.229,A -85,B 0,C 180,E1 -11570.25,E2 -11570.25} C_VEL
LIN {X 0,Y 395.326,Z 223.927,A -85,B 0,C 180,E1 -11573.13,E2 -11573.13} C_VEL
LIN {X 0,Y 397.231,Z 229.325,A -85,B 0,C 180,E1 -11574.084,E2 -11574.084} C_VEL
LIN {X 0,Y 405.135,Z 244.505,A -85,B 0,C 180,E1 -11575.284,E2 -11575.284} C_VEL
LIN {X 0,Y 411.421,Z 257.652,A -85,B 0,C 180,E1 -11576.207,E2 -11576.207} C_VEL
LIN {X 0,Y 413.236,Z 269.614,A -85,B 0,C 180,E1 -11576.643,E2 -11576.643} C_VEL
LIN {X 0,Y 408.559,Z 437.247,A -85,B 0,C 180,E1 -11579.783,E2 -11579.783} C_VEL
LIN {X 0,Y 407.409,Z 453.892,A -85,B 0,C 180,E1 -11580.268,E2 -11580.268} C_VEL
LIN {X 0,Y 406.085,Z 470.03,A -85,B 0,C 180,E1 -11580.944,E2 -11580.944} C_VEL
LIN {X 0,Y 404.276,Z 486.868,A -85,B 0,C 180,E1 -11581.866,E2 -11581.866} C_VEL
LIN {X 0,Y 402.351,Z 502.905,A -85,B 0,C 180,E1 -11582.99,E2 -11582.99} C_VEL
LIN {X 0,Y 400.372,Z 517.568,A -85,B 0,C 180,E1 -11584.25,E2 -11584.25} C_VEL
LIN {X 0,Y 398.422,Z 531.134,A -85,B 0,C 180,E1 -11585.65,E2 -11585.65} C_VEL
LIN {X 0,Y 396.528,Z 543.485,A -85,B 0,C 180,E1 -11587.166,E2 -11587.166} C_VEL
LIN {X 0,Y 394.693,Z 555.286,A -85,B 0,C 180,E1 -11588.865,E2 -11588.865} C_VEL
LIN {X 0,Y 393.121,Z 566.062,A -85,B 0,C 180,E1 -11590.687,E2 -11590.687} C_VEL
LIN {X 0,Y 391.839,Z 575.242,A -85,B 0,C 180,E1 -11592.517,E2 -11592.517} C_VEL
LIN {X 0,Y 390.627,Z 584.162,A -85,B 0,C 180,E1 -11594.611,E2 -11594.611} C_VEL
LIN {X 0,Y 389.75,Z 592.051,A -85,B 0,C 180,E1 -11596.837,E2 -11596.837} C_VEL
LIN {X 0,Y 389.194,Z 598.534,A -85,B 0,C 180,E1 -11599.071,E2 -11599.071} C_VEL
LIN {X 0,Y 388.84,Z 604.411,A -85,B 0,C 180,E1 -11601.687,E2 -11601.687} C_VEL
LIN {X 0,Y 388.723,Z 608.058,A -85,B 0,C 180,E1 -11603.923,E2 -11603.923} C_VEL
LIN {X 0,Y 388.648,Z 610.335,A -85,B 0,C 180,E1 -11605.852,E2 -11605.852} C_VEL
LIN {X 0,Y 388.675,Z 611.743,A -85,B 0,C 180,E1 -11607.928,E2 -11607.928} C_VEL
LIN {X 0,Y 388.704,Z 612.259,A -85,B 0,C 180,E1 -11610,E2 -11610} C_VEL
LIN {X 0,Y 388.676,Z 611.712,A -85,B 0,C 180,E1 -11612.073,E2 -11612.073} C_VEL
LIN {X 0,Y 388.648,Z 610.265,A -85,B 0,C 180,E1 -11614.148,E2 -11614.148} C_VEL
LIN {X 0,Y 388.747,Z 607.739,A -85,B 0,C 180,E1 -11616.227,E2 -11616.227} C_VEL
LIN {X 0,Y 388.841,Z 604.237,A -85,B 0,C 180,E1 -11618.314,E2 -11618.314} C_VEL
LIN {X 0,Y 389.034,Z 599.589,A -85,B 0,C 180,E1 -11620.408,E2 -11620.408} C_VEL
LIN {X 0,Y 389.622,Z 593.795,A -85,B 0,C 180,E1 -11622.501,E2 -11622.501} C_VEL
LIN {X 0,Y 390.261,Z 586.764,A -85,B 0,C 180,E1 -11624.603,E2 -11624.603} C_VEL
LIN {X 0,Y 391.506,Z 577.088,A -85,B 0,C 180,E1 -11626.96,E2 -11626.96} C_VEL
LIN {X 0,Y 392.806,Z 566.675,A -85,B 0,C 180,E1 -11629.058,E2 -11629.058} C_VEL
LIN {X 0,Y 394.359,Z 555.911,A -85,B 0,C 180,E1 -11630.881,E2 -11630.881} C_VEL
LIN {X 0,Y 396.075,Z 544.363,A -85,B 0,C 180,E1 -11632.55,E2 -11632.55} C_VEL
LIN {X 0,Y 397.714,Z 532.83,A -85,B 0,C 180,E1 -11633.981,E2 -11633.981} C_VEL
LIN {X 0,Y 399.588,Z 519.377,A -85,B 0,C 180,E1 -11635.386,E2 -11635.386} C_VEL
LIN {X 0,Y 401.495,Z 504.769,A -85,B 0,C 180,E1 -11636.66,E2 -11636.66} C_VEL
LIN {X 0,Y 403.164,Z 491.037,A -85,B 0,C 180,E1 -11637.654,E2 -11637.654} C_VEL
LIN {X 0,Y 404.856,Z 475.068,A -85,B 0,C 180,E1 -11638.585,E2 -11638.585} C_VEL
LIN {X 0,Y 406.167,Z 458.413,A -85,B 0,C 180,E1 -11639.334,E2 -11639.334} C_VEL
LIN {X 0,Y 407.263,Z 442.181,A -85,B 0,C 180,E1 -11639.851,E2 -11639.851} C_VEL
LIN {X 0,Y 408.084,Z 422.244,A -85,B 0,C 180,E1 -11640.265,E2 -11640.265} C_VEL
LIN {X 0,Y 411.897,Z 268.752,A -85,B 0,C 180,E1 -11643.093,E2 -11643.093} C_VEL
LIN {X 0,Y 409.742,Z 256.231,A -85,B 0,C 180,E1 -11643.541,E2 -11643.541} C_VEL
LIN {X 0,Y 398.975,Z 233.876,A -85,B 0,C 180,E1 -11645.002,E2 -11645.002} C_VEL
LIN {X 0,Y 397.113,Z 230.041,A -85,B 0,C 180,E1 -11645.268,E2 -11645.268} C_VEL
LIN {X 0,Y 390.832,Z 211.576,A -85,B 0,C 180,E1 -11648.517,E2 -11648.517} C_VEL
LIN {X 0,Y 390.077,Z 209.211,A -85,B 0,C 180,E1 -11648.944,E2 -11648.944} C_VEL
LIN {X 0,Y 390.037,Z 209.207,A -85,B 0,C 180,E1 -11652.373,E2 -11652.373} C_VEL
LIN {X 0,Y 390.041,Z 209.204,A -85,B 0,C 180,E1 -11655.354,E2 -11655.354} C_VEL
LIN {X 0,Y 390.021,Z 209.215,A -85,B 0,C 180,E1 -11658.186,E2 -11658.186} C_VEL
LIN {X 0,Y 390.063,Z 209.21,A -85,B 0,C 180,E1 -11660.905,E2 -11660.905} C_VEL
LIN {X 0,Y 390.082,Z 209.201,A -85,B 0,C 180,E1 -11664.793,E2 -11664.793} C_VEL
LIN {X 0,Y 390.02,Z 209.199,A -85,B 0,C 180,E1 -11668.496,E2 -11668.496} C_VEL
LIN {X 0,Y 390.115,Z 209.202,A -85,B 0,C 180,E1 -11672.07,E2 -11672.07} C_VEL
LIN {X 0,Y 390.077,Z 209.202,A -85,B 0,C 180,E1 -11675.519,E2 -11675.519} C_VEL
LIN {X 0,Y 390.053,Z 209.202,A -85,B 0,C 180,E1 -11678.878,E2 -11678.878} C_VEL
LIN {X 0,Y 390.108,Z 209.189,A -85,B 0,C 180,E1 -11682.166,E2 -11682.166} C_VEL
LIN {X 0,Y 390.141,Z 209.195,A -85,B 0,C 180,E1 -11685.393,E2 -11685.393} C_VEL
LIN {X 0,Y 390.144,Z 209.171,A -85,B 0,C 180,E1 -11688.571,E2 -11688.571} C_VEL
LIN {X 0,Y 390.267,Z 209.183,A -85,B 0,C 180,E1 -11692.071,E2 -11692.071} C_VEL
LIN {X 0,Y 390.219,Z 209.176,A -85,B 0,C 180,E1 -11694.833,E2 -11694.833} C_VEL
LIN {X 0,Y 390.415,Z 209.134,A -85,B 0,C 180,E1 -11697.937,E2 -11697.937} C_VEL
LIN {X 0,Y 390.545,Z 209.141,A -85,B 0,C 180,E1 -11700,E2 -11700} C_VEL
LIN {X 0,Y 390.306,Z 209.173,A -85,B 0,C 180,E1 -11703.097,E2 -11703.097} C_VEL
LIN {X 0,Y 390.299,Z 209.168,A -85,B 0,C 180,E1 -11706.65,E2 -11706.65} C_VEL
LIN {X 0,Y 390.202,Z 209.189,A -85,B 0,C 180,E1 -11709.329,E2 -11709.329} C_VEL
LIN {X 0,Y 390.192,Z 209.182,A -85,B 0,C 180,E1 -11713.438,E2 -11713.438} C_VEL
LIN {X 0,Y 390.146,Z 209.192,A -85,B 0,C 180,E1 -11717.308,E2 -11717.308} C_VEL
LIN {X 0,Y 390.085,Z 209.203,A -85,B 0,C 180,E1 -11720.47,E2 -11720.47} C_VEL
LIN {X 0,Y 390.087,Z 209.204,A -85,B 0,C 180,E1 -11723.351,E2 -11723.351} C_VEL
LIN {X 0,Y 390.111,Z 209.194,A -85,B 0,C 180,E1 -11726.768,E2 -11726.768} C_VEL
LIN {X 0,Y 390.042,Z 209.205,A -85,B 0,C 180,E1 -11730.299,E2 -11730.299} C_VEL
LIN {X 0,Y 390.067,Z 209.209,A -85,B 0,C 180,E1 -11734.025,E2 -11734.025} C_VEL
LIN {X 0,Y 390.044,Z 209.2,A -85,B 0,C 180,E1 -11737.551,E2 -11737.551} C_VEL
LIN {X 0,Y 390.055,Z 209.209,A -85,B 0,C 180,E1 -11740.822,E2 -11740.822} C_VEL
LIN {X 0,Y 390.052,Z 209.199,A -85,B 0,C 180,E1 -11743.886,E2 -11743.886} C_VEL
LIN {X 0,Y 390.055,Z 209.209,A -85,B 0,C 180,E1 -11746.79,E2 -11746.79} C_VEL
LIN {X 0,Y 390.055,Z 209.202,A -85,B 0,C 180,E1 -11749.561,E2 -11749.561} C_VEL
LIN {X 0,Y 390.041,Z 209.209,A -85,B 0,C 180,E1 -11752.45,E2 -11752.45} C_VEL
LIN {X 0,Y 390.067,Z 209.209,A -85,B 0,C 180,E1 -11755.975,E2 -11755.975} C_VEL
LIN {X 0,Y 390.046,Z 209.212,A -85,B 0,C 180,E1 -11759.869,E2 -11759.869} C_VEL
LIN {X 0,Y 390.113,Z 209.197,A -85,B 0,C 180,E1 -11763.232,E2 -11763.232} C_VEL
LIN {X 0,Y 390.106,Z 209.197,A -85,B 0,C 180,E1 -11766.75,E2 -11766.75} C_VEL
LIN {X 0,Y 390.103,Z 209.186,A -85,B 0,C 180,E1 -11769.983,E2 -11769.983} C_VEL
LIN {X 0,Y 390.138,Z 209.202,A -85,B 0,C 180,E1 -11773.248,E2 -11773.248} C_VEL
LIN {X 0,Y 390.194,Z 209.172,A -85,B 0,C 180,E1 -11776.561,E2 -11776.561} C_VEL
LIN {X 0,Y 390.191,Z 209.319,A -85,B 0,C 180,E1 -11779.83,E2 -11779.83} C_VEL
LIN {X 0,Y 390.844,Z 211.387,A -85,B 0,C 180,E1 -11780.19,E2 -11780.19} C_VEL
LIN {X 0,Y 401.293,Z 230.494,A -85,B 0,C 180,E1 -11781.627,E2 -11781.627} C_VEL
LIN {X 0,Y 412.056,Z 252.438,A -85,B 0,C 180,E1 -11783.066,E2 -11783.066} C_VEL
LIN {X 0,Y 407.873,Z 416.594,A -85,B 0,C 180,E1 -11786.109,E2 -11786.109} C_VEL
LIN {X 0,Y 406.969,Z 433.007,A -85,B 0,C 180,E1 -11786.597,E2 -11786.597} C_VEL
LIN {X 0,Y 405.753,Z 449.162,A -85,B 0,C 180,E1 -11787.27,E2 -11787.27} C_VEL
LIN {X 0,Y 404.384,Z 464.854,A -85,B 0,C 180,E1 -11788.132,E2 -11788.132} C_VEL
LIN {X 0,Y 404.196,Z 466.597,A -85,B 0,C 180,E1 -11788.242,E2 -11788.242} C_VEL
LIN {X 0,Y 403.026,Z 472.05,A -85,B 0,C 180,E1 -11788.552,E2 -11788.552} C_VEL
LIN {X 0,Y 396.47,Z 487.632,A -85,B 0,C 180,E1 -11789.403,E2 -11789.403} C_VEL
LIN {X 0,Y 394.864,Z 492.56,A -85,B 0,C 180,E1 -11789.776,E2 -11789.776} C_VEL
LIN {X 0,Y 394.56,Z 494.195,A -85,B 0,C 180,E1 -11789.918,E2 -11789.918} C_VEL
LIN {X 0,Y 392.641,Z 507.595,A -85,B 0,C 180,E1 -11791.282,E2 -11791.282} C_VEL
LIN {X 0,Y 390.763,Z 520.43,A -85,B 0,C 180,E1 -11792.835,E2 -11792.835} C_VEL
LIN {X 0,Y 388.773,Z 533.003,A -85,B 0,C 180,E1 -11794.635,E2 -11794.635} C_VEL
LIN {X 0,Y 387.021,Z 544.07,A -85,B 0,C 180,E1 -11796.516,E2 -11796.516} C_VEL
LIN {X 0,Y 385.445,Z 554.535,A -85,B 0,C 180,E1 -11798.651,E2 -11798.651} C_VEL
LIN {X 0,Y 384.215,Z 563.32,A -85,B 0,C 180,E1 -11800.806,E2 -11800.806} C_VEL
LIN {X 0,Y 383.176,Z 571.05,A -85,B 0,C 180,E1 -11803.1,E2 -11803.1} C_VEL
LIN {X 0,Y 382.384,Z 577.463,A -85,B 0,C 180,E1 -11805.456,E2 -11805.456} C_VEL
LIN {X 0,Y 381.989,Z 582.218,A -85,B 0,C 180,E1 -11807.672,E2 -11807.672} C_VEL
LIN {X 0,Y 381.59,Z 585.996,A -85,B 0,C 180,E1 -11810.066,E2 -11810.066} C_VEL
LIN {X 0,Y 381.43,Z 587.793,A -85,B 0,C 180,E1 -11811.623,E2 -11811.623} C_VEL
LIN {X 0,Y 381.304,Z 589.449,A -85,B 0,C 180,E1 -11813.921,E2 -11813.921} C_VEL
LIN {X 0,Y 381.301,Z 590.027,A -85,B 0,C 180,E1 -11816.254,E2 -11816.254} C_VEL
LIN {X 0,Y 381.385,Z 589.37,A -85,B 0,C 180,E1 -11818.627,E2 -11818.627} C_VEL
LIN {X 0,Y 381.53,Z 587.466,A -85,B 0,C 180,E1 -11821.049,E2 -11821.049} C_VEL
LIN {X 0,Y 381.864,Z 584.236,A -85,B 0,C 180,E1 -11823.513,E2 -11823.513} C_VEL
LIN {X 0,Y 382.243,Z 580.834,A -85,B 0,C 180,E1 -11825.391,E2 -11825.391} C_VEL
LIN {X 0,Y 382.856,Z 575.044,A -85,B 0,C 180,E1 -11827.876,E2 -11827.876} C_VEL
LIN {X 0,Y 383.726,Z 568.156,A -85,B 0,C 180,E1 -11830.21,E2 -11830.21} C_VEL
LIN {X 0,Y 384.948,Z 559.873,A -85,B 0,C 180,E1 -11832.493,E2 -11832.493} C_VEL
LIN {X 0,Y 386.329,Z 551.284,A -85,B 0,C 180,E1 -11834.457,E2 -11834.457} C_VEL
LIN {X 0,Y 387.989,Z 541.06,A -85,B 0,C 180,E1 -11836.431,E2 -11836.431} C_VEL
LIN {X 0,Y 389.918,Z 529.777,A -85,B 0,C 180,E1 -11838.27,E2 -11838.27} C_VEL
LIN {X 0,Y 392.006,Z 517.197,A -85,B 0,C 180,E1 -11840.003,E2 -11840.003} C_VEL
LIN {X 0,Y 393.959,Z 504.821,A -85,B 0,C 180,E1 -11841.443,E2 -11841.443} C_VEL
LIN {X 0,Y 395.881,Z 491.302,A -85,B 0,C 180,E1 -11842.766,E2 -11842.766} C_VEL
LIN {X 0,Y 397.908,Z 475.87,A -85,B 0,C 180,E1 -11844.012,E2 -11844.012} C_VEL
LIN {X 0,Y 399.662,Z 460.293,A -85,B 0,C 180,E1 -11845.028,E2 -11845.028} C_VEL
LIN {X 0,Y 401.079,Z 444.858,A -85,B 0,C 180,E1 -11845.826,E2 -11845.826} C_VEL
LIN {X 0,Y 402.31,Z 428.295,A -85,B 0,C 180,E1 -11846.457,E2 -11846.457} C_VEL
LIN {X 0,Y 403.139,Z 411.121,A -85,B 0,C 180,E1 -11846.899,E2 -11846.899} C_VEL
LIN {X 0,Y 407.626,Z 255.943,A -85,B 0,C 180,E1 -11849.847,E2 -11849.847} C_VEL
LIN {X 0,Y 399.08,Z 238.855,A -85,B 0,C 180,E1 -11851.129,E2 -11851.129} C_VEL
LIN {X 0,Y 390.803,Z 224.176,A -85,B 0,C 180,E1 -11852.414,E2 -11852.414} C_VEL
LIN {X 0,Y 385.689,Z 215.908,A -85,B 0,C 180,E1 -11853.235,E2 -11853.235} C_VEL
LIN {X 0,Y 383.736,Z 212.445,A -85,B 0,C 180,E1 -11853.6,E2 -11853.6} C_VEL
LIN {X 0,Y 383.031,Z 210.088,A -85,B 0,C 180,E1 -11854.15,E2 -11854.15} C_VEL
LIN {X 0,Y 382.982,Z 210.087,A -85,B 0,C 180,E1 -11857.334,E2 -11857.334} C_VEL
LIN {X 0,Y 383.052,Z 210.077,A -85,B 0,C 180,E1 -11860.716,E2 -11860.716} C_VEL
LIN {X 0,Y 383.073,Z 210.071,A -85,B 0,C 180,E1 -11864.026,E2 -11864.026} C_VEL
LIN {X 0,Y 383.13,Z 210.065,A -85,B 0,C 180,E1 -11867.284,E2 -11867.284} C_VEL
LIN {X 0,Y 383.137,Z 210.073,A -85,B 0,C 180,E1 -11870.498,E2 -11870.498} C_VEL
LIN {X 0,Y 383.265,Z 210.053,A -85,B 0,C 180,E1 -11873.683,E2 -11873.683} C_VEL
LIN {X 0,Y 383.379,Z 210.04,A -85,B 0,C 180,E1 -11877.899,E2 -11877.899} C_VEL
LIN {X 0,Y 383.513,Z 210.026,A -85,B 0,C 180,E1 -11880,E2 -11880} C_VEL
LIN {X 0,Y 383.24,Z 210.054,A -85,B 0,C 180,E1 -11883.154,E2 -11883.154} C_VEL
LIN {X 0,Y 383.277,Z 210.054,A -85,B 0,C 180,E1 -11886.316,E2 -11886.316} C_VEL
LIN {X 0,Y 383.145,Z 210.07,A -85,B 0,C 180,E1 -11889.502,E2 -11889.502} C_VEL
LIN {X 0,Y 383.119,Z 210.072,A -85,B 0,C 180,E1 -11893.536,E2 -11893.536} C_VEL
LIN {X 0,Y 383.089,Z 210.077,A -85,B 0,C 180,E1 -11897.455,E2 -11897.455} C_VEL
LIN {X 0,Y 383.023,Z 210.085,A -85,B 0,C 180,E1 -11900.647,E2 -11900.647} C_VEL
LIN {X 0,Y 383.028,Z 210.084,A -85,B 0,C 180,E1 -11903.808,E2 -11903.808} C_VEL
LIN {X 0,Y 383.074,Z 210.077,A -85,B 0,C 180,E1 -11906.124,E2 -11906.124} C_VEL
LIN {X 0,Y 382.986,Z 210.092,A -85,B 0,C 180,E1 -11909.7,E2 -11909.7} C_VEL
LIN {X 0,Y 382.998,Z 210.091,A -85,B 0,C 180,E1 -11913.401,E2 -11913.401} C_VEL
LIN {X 0,Y 383.027,Z 210.088,A -85,B 0,C 180,E1 -11916.165,E2 -11916.165} C_VEL
LIN {X 0,Y 383.004,Z 210.092,A -85,B 0,C 180,E1 -11919.959,E2 -11919.959} C_VEL
LIN {X 0,Y 383,Z 210.096,A -85,B 0,C 180,E1 -11922.779,E2 -11922.779} C_VEL
LIN {X 0,Y 382.992,Z 210.095,A -85,B 0,C 180,E1 -11925.79,E2 -11925.79} C_VEL
LIN {X 0,Y 383.026,Z 210.136,A -85,B 0,C 180,E1 -11929.474,E2 -11929.474} C_VEL
LIN {X 0,Y 388.389,Z 225.013,A -85,B 0,C 180,E1 -11932.501,E2 -11932.501} C_VEL
LIN {X 0,Y 389.821,Z 228.952,A -85,B 0,C 180,E1 -11933.223,E2 -11933.223} C_VEL
LIN {X 0,Y 397.752,Z 243.701,A -85,B 0,C 180,E1 -11934.476,E2 -11934.476} C_VEL
LIN {X 0,Y 405.834,Z 260.369,A -85,B 0,C 180,E1 -11935.709,E2 -11935.709} C_VEL
LIN {X 0,Y 407.393,Z 271.607,A -85,B 0,C 180,E1 -11936.113,E2 -11936.113} C_VEL
LIN {X 0,Y 402.52,Z 437.146,A -85,B 0,C 180,E1 -11939.262,E2 -11939.262} C_VEL
LIN {X 0,Y 401.343,Z 453.314,A -85,B 0,C 180,E1 -11939.736,E2 -11939.736} C_VEL
LIN {X 0,Y 400.018,Z 468.904,A -85,B 0,C 180,E1 -11940.388,E2 -11940.388} C_VEL
LIN {X 0,Y 398.266,Z 484.962,A -85,B 0,C 180,E1 -11941.259,E2 -11941.259} C_VEL
LIN {X 0,Y 396.437,Z 499.746,A -85,B 0,C 180,E1 -11942.267,E2 -11942.267} C_VEL
LIN {X 0,Y 394.312,Z 514.843,A -85,B 0,C 180,E1 -11943.54,E2 -11943.54} C_VEL
LIN {X 0,Y 392.228,Z 528.714,A -85,B 0,C 180,E1 -11944.957,E2 -11944.957} C_VEL
LIN {X 0,Y 390.334,Z 540.594,A -85,B 0,C 180,E1 -11946.384,E2 -11946.384} C_VEL
LIN {X 0,Y 388.539,Z 551.811,A -85,B 0,C 180,E1 -11947.956,E2 -11947.956} C_VEL
LIN {X 0,Y 386.766,Z 562.995,A -85,B 0,C 180,E1 -11949.803,E2 -11949.803} C_VEL
LIN {X 0,Y 385.371,Z 571.855,A -85,B 0,C 180,E1 -11951.499,E2 -11951.499} C_VEL
LIN {X 0,Y 384.158,Z 580.878,A -85,B 0,C 180,E1 -11953.527,E2 -11953.527} C_VEL
LIN {X 0,Y 383.092,Z 588.829,A -85,B 0,C 180,E1 -11955.661,E2 -11955.661} C_VEL
LIN {X 0,Y 382.407,Z 595.473,A -85,B 0,C 180,E1 -11957.799,E2 -11957.799} C_VEL
LIN {X 0,Y 381.885,Z 600.884,A -85,B 0,C 180,E1 -11959.932,E2 -11959.932} C_VEL
LIN {X 0,Y 381.745,Z 604.223,A -85,B 0,C 180,E1 -11961.531,E2 -11961.531} C_VEL
LIN {X 0,Y 381.648,Z 608.041,A -85,B 0,C 180,E1 -11963.933,E2 -11963.933} C_VEL
LIN {X 0,Y 381.573,Z 610.138,A -85,B 0,C 180,E1 -11965.775,E2 -11965.775} C_VEL
LIN {X 0,Y 381.572,Z 611.543,A -85,B 0,C 180,E1 -11967.889,E2 -11967.889} C_VEL
LIN {X 0,Y 381.635,Z 612.052,A -85,B 0,C 180,E1 -11970,E2 -11970} C_VEL
LIN {X 0,Y 381.573,Z 611.5,A -85,B 0,C 180,E1 -11972.111,E2 -11972.111} C_VEL
LIN {X 0,Y 381.573,Z 610.045,A -85,B 0,C 180,E1 -11974.225,E2 -11974.225} C_VEL
LIN {X 0,Y 381.658,Z 607.513,A -85,B 0,C 180,E1 -11976.344,E2 -11976.344} C_VEL
LIN {X 0,Y 381.746,Z 603.999,A -85,B 0,C 180,E1 -11978.47,E2 -11978.47} C_VEL
LIN {X 0,Y 381.995,Z 599.345,A -85,B 0,C 180,E1 -11980.602,E2 -11980.602} C_VEL
LIN {X 0,Y 382.587,Z 593.536,A -85,B 0,C 180,E1 -11982.735,E2 -11982.735} C_VEL
LIN {X 0,Y 383.272,Z 586.493,A -85,B 0,C 180,E1 -11984.875,E2 -11984.875} C_VEL
LIN {X 0,Y 384.577,Z 576.8,A -85,B 0,C 180,E1 -11987.275,E2 -11987.275} C_VEL
LIN {X 0,Y 385.994,Z 566.365,A -85,B 0,C 180,E1 -11989.408,E2 -11989.408} C_VEL
LIN {X 0,Y 387.615,Z 555.566,A -85,B 0,C 180,E1 -11991.262,E2 -11991.262} C_VEL
LIN {X 0,Y 389.442,Z 543.512,A -85,B 0,C 180,E1 -11993.021,E2 -11993.021} C_VEL
LIN {X 0,Y 391.366,Z 531.284,A -85,B 0,C 180,E1 -11994.536,E2 -11994.536} C_VEL
LIN {X 0,Y 393.105,Z 518.927,A -85,B 0,C 180,E1 -11995.835,E2 -11995.835} C_VEL
LIN {X 0,Y 395.06,Z 504.261,A -85,B 0,C 180,E1 -11997.129,E2 -11997.129} C_VEL
LIN {X 0,Y 397.05,Z 488.457,A -85,B 0,C 180,E1 -11998.261,E2 -11998.261} C_VEL
LIN {X 0,Y 398.687,Z 473.126,A -85,B 0,C 180,E1 -11999.141,E2 -11999.141} C_VEL
LIN {X 0,Y 400.005,Z 456.869,A -85,B 0,C 180,E1 -11999.867,E2 -11999.867} C_VEL
LIN {X 0,Y 401.174,Z 439.997,A -85,B 0,C 180,E1 -12000.388,E2 -12000.388} C_VEL
LIN {X 0,Y 401.948,Z 418.551,A -85,B 0,C 180,E1 -12000.822,E2 -12000.822} C_VEL
LIN {X 0,Y 405.912,Z 270.68,A -85,B 0,C 180,E1 -12003.575,E2 -12003.575} C_VEL
LIN {X 0,Y 404.053,Z 259.258,A -85,B 0,C 180,E1 -12003.984,E2 -12003.984} C_VEL
LIN {X 0,Y 393.687,Z 237.602,A -85,B 0,C 180,E1 -12005.428,E2 -12005.428} C_VEL
LIN {X 0,Y 389.65,Z 229.587,A -85,B 0,C 180,E1 -12006.036,E2 -12006.036} C_VEL
LIN {X 0,Y 384.367,Z 214.089,A -85,B 0,C 180,E1 -12008.834,E2 -12008.834} C_VEL
LIN {X 0,Y 383.001,Z 210.085,A -85,B 0,C 180,E1 -12009.613,E2 -12009.613} C_VEL
LIN {X 0,Y 383.004,Z 210.082,A -85,B 0,C 180,E1 -12012.779,E2 -12012.779} C_VEL
LIN {X 0,Y 382.994,Z 210.08,A -85,B 0,C 180,E1 -12015.789,E2 -12015.789} C_VEL
LIN {X 0,Y 382.968,Z 210.086,A -85,B 0,C 180,E1 -12018.799,E2 -12018.799} C_VEL
LIN {X 0,Y 382.994,Z 210.091,A -85,B 0,C 180,E1 -12022.097,E2 -12022.097} C_VEL
LIN {X 0,Y 383.015,Z 210.089,A -85,B 0,C 180,E1 -12025.332,E2 -12025.332} C_VEL
LIN {X 0,Y 382.98,Z 210.079,A -85,B 0,C 180,E1 -12029.081,E2 -12029.081} C_VEL
LIN {X 0,Y 383.054,Z 210.072,A -85,B 0,C 180,E1 -12032.698,E2 -12032.698} C_VEL
LIN {X 0,Y 383.049,Z 210.069,A -85,B 0,C 180,E1 -12035.04,E2 -12035.04} C_VEL
LIN {X 0,Y 382.99,Z 210.087,A -85,B 0,C 180,E1 -12038.469,E2 -12038.469} C_VEL
LIN {X 0,Y 383.05,Z 210.066,A -85,B 0,C 180,E1 -12041.826,E2 -12041.826} C_VEL
LIN {X 0,Y 383.107,Z 210.073,A -85,B 0,C 180,E1 -12045.118,E2 -12045.118} C_VEL
LIN {X 0,Y 383.093,Z 210.048,A -85,B 0,C 180,E1 -12048.358,E2 -12048.358} C_VEL
LIN {X 0,Y 383.225,Z 210.06,A -85,B 0,C 180,E1 -12052.014,E2 -12052.014} C_VEL
LIN {X 0,Y 383.191,Z 210.052,A -85,B 0,C 180,E1 -12054.738,E2 -12054.738} C_VEL
LIN {X 0,Y 383.382,Z 210.009,A -85,B 0,C 180,E1 -12057.899,E2 -12057.899} C_VEL
LIN {X 0,Y 383.515,Z 210.017,A -85,B 0,C 180,E1 -12060,E2 -12060} C_VEL
LIN {X 0,Y 383.243,Z 210.053,A -85,B 0,C 180,E1 -12063.154,E2 -12063.154} C_VEL
LIN {X 0,Y 383.258,Z 210.045,A -85,B 0,C 180,E1 -12066.643,E2 -12066.643} C_VEL
LIN {X 0,Y 383.148,Z 210.068,A -85,B 0,C 180,E1 -12069.502,E2 -12069.502} C_VEL
LIN {X 0,Y 383.123,Z 210.063,A -85,B 0,C 180,E1 -12073.536,E2 -12073.536} C_VEL
LIN {X 0,Y 383.093,Z 210.069,A -85,B 0,C 180,E1 -12077.455,E2 -12077.455} C_VEL
LIN {X 0,Y 383.026,Z 210.081,A -85,B 0,C 180,E1 -12080.647,E2 -12080.647} C_VEL
LIN {X 0,Y 383.031,Z 210.078,A -85,B 0,C 180,E1 -12083.807,E2 -12083.807} C_VEL
LIN {X 0,Y 383.078,Z 210.065,A -85,B 0,C 180,E1 -12086.123,E2 -12086.123} C_VEL
LIN {X 0,Y 383.047,Z 210.082,A -85,B 0,C 180,E1 -12088.492,E2 -12088.492} C_VEL
LIN {X 0,Y 383.009,Z 210.073,A -85,B 0,C 180,E1 -12092.15,E2 -12092.15} C_VEL
LIN {X 0,Y 383.016,Z 210.085,A -85,B 0,C 180,E1 -12094.668,E2 -12094.668} C_VEL
LIN {X 0,Y 383,Z 210.075,A -85,B 0,C 180,E1 -12097.904,E2 -12097.904} C_VEL
LIN {X 0,Y 382.983,Z 210.093,A -85,B 0,C 180,E1 -12101.347,E2 -12101.347} C_VEL
LIN {X 0,Y 382.994,Z 210.08,A -85,B 0,C 180,E1 -12104.303,E2 -12104.303} C_VEL
LIN {X 0,Y 383.009,Z 210.089,A -85,B 0,C 180,E1 -12107.24,E2 -12107.24} C_VEL
LIN {X 0,Y 383.012,Z 210.084,A -85,B 0,C 180,E1 -12110.414,E2 -12110.414} C_VEL
LIN {X 0,Y 383.023,Z 210.074,A -85,B 0,C 180,E1 -12114.044,E2 -12114.044} C_VEL
LIN {X 0,Y 382.985,Z 210.085,A -85,B 0,C 180,E1 -12117.578,E2 -12117.578} C_VEL
LIN {X 0,Y 382.991,Z 210.09,A -85,B 0,C 180,E1 -12120.3,E2 -12120.3} C_VEL
LIN {X 0,Y 383.08,Z 210.078,A -85,B 0,C 180,E1 -12124.021,E2 -12124.021} C_VEL
LIN {X 0,Y 383.013,Z 210.087,A -85,B 0,C 180,E1 -12127.335,E2 -12127.335} C_VEL
LIN {X 0,Y 383.059,Z 210.055,A -85,B 0,C 180,E1 -12130.716,E2 -12130.716} C_VEL
LIN {X 0,Y 383.08,Z 210.082,A -85,B 0,C 180,E1 -12134.027,E2 -12134.027} C_VEL
LIN {X 0,Y 383.136,Z 210.059,A -85,B 0,C 180,E1 -12137.284,E2 -12137.284} C_VEL
LIN {X 0,Y 383.129,Z 210.14,A -85,B 0,C 180,E1 -12139.196,E2 -12139.196} C_VEL
LIN {X 0,Y 383.534,Z 211.7,A -85,B 0,C 180,E1 -12139.441,E2 -12139.441} C_VEL
LIN {X 0,Y 390.978,Z 224.858,A -85,B 0,C 180,E1 -12140.508,E2 -12140.508} C_VEL
LIN {X 0,Y 399.339,Z 240.919,A -85,B 0,C 180,E1 -12141.671,E2 -12141.671} C_VEL
LIN {X 0,Y 406.03,Z 254.8,A -85,B 0,C 180,E1 -12142.582,E2 -12142.582} C_VEL
LIN {X 0,Y 401.649,Z 417.169,A -85,B 0,C 180,E1 -12145.634,E2 -12145.634} C_VEL
LIN {X 0,Y 400.704,Z 433.636,A -85,B 0,C 180,E1 -12146.134,E2 -12146.134} C_VEL
LIN {X 0,Y 399.387,Z 450.311,A -85,B 0,C 180,E1 -12146.847,E2 -12146.847} C_VEL
LIN {X 0,Y 397.956,Z 465.796,A -85,B 0,C 180,E1 -12147.722,E2 -12147.722} C_VEL
LIN {X 0,Y 396.338,Z 480.239,A -85,B 0,C 180,E1 -12148.73,E2 -12148.73} C_VEL
LIN {X 0,Y 394.56,Z 494.195,A -85,B 0,C 180,E1 -12149.918,E2 -12149.918} C_VEL
LIN {X 0,Y 393.253,Z 499.178,A -85,B 0,C 180,E1 -12150.341,E2 -12150.341} C_VEL
LIN {X 0,Y 389.462,Z 507.192,A -85,B 0,C 180,E1 -12150.995,E2 -12150.995} C_VEL
LIN {X 0,Y 385.669,Z 514.877,A -85,B 0,C 180,E1 -12151.726,E2 -12151.726} C_VEL
LIN {X 0,Y 384.373,Z 519.339,A -85,B 0,C 180,E1 -12152.266,E2 -12152.266} C_VEL
LIN {X 0,Y 382.377,Z 531.217,A -85,B 0,C 180,E1 -12153.952,E2 -12153.952} C_VEL
LIN {X 0,Y 380.53,Z 542.339,A -85,B 0,C 180,E1 -12155.83,E2 -12155.83} C_VEL
LIN {X 0,Y 379.057,Z 551.866,A -85,B 0,C 180,E1 -12157.725,E2 -12157.725} C_VEL
LIN {X 0,Y 377.63,Z 561.169,A -85,B 0,C 180,E1 -12159.912,E2 -12159.912} C_VEL
LIN {X 0,Y 376.383,Z 569.828,A -85,B 0,C 180,E1 -12162.399,E2 -12162.399} C_VEL
LIN {X 0,Y 375.526,Z 576.107,A -85,B 0,C 180,E1 -12164.634,E2 -12164.634} C_VEL
LIN {X 0,Y 374.976,Z 581.542,A -85,B 0,C 180,E1 -12167.086,E2 -12167.086} C_VEL
LIN {X 0,Y 374.713,Z 584.208,A -85,B 0,C 180,E1 -12168.593,E2 -12168.593} C_VEL
LIN {X 0,Y 374.395,Z 587.306,A -85,B 0,C 180,E1 -12170.895,E2 -12170.895} C_VEL
LIN {X 0,Y 374.241,Z 589.333,A -85,B 0,C 180,E1 -12173.226,E2 -12173.226} C_VEL
LIN {X 0,Y 374.222,Z 590.17,A -85,B 0,C 180,E1 -12175.651,E2 -12175.651} C_VEL
LIN {X 0,Y 374.302,Z 589.849,A -85,B 0,C 180,E1 -12178.057,E2 -12178.057} C_VEL
LIN {X 0,Y 374.407,Z 588.393,A -85,B 0,C 180,E1 -12180.451,E2 -12180.451} C_VEL
LIN {X 0,Y 374.681,Z 585.518,A -85,B 0,C 180,E1 -12182.953,E2 -12182.953} C_VEL
LIN {X 0,Y 374.979,Z 583.184,A -85,B 0,C 180,E1 -12184.446,E2 -12184.446} C_VEL
LIN {X 0,Y 375.436,Z 578.464,A -85,B 0,C 180,E1 -12186.799,E2 -12186.799} C_VEL
LIN {X 0,Y 376.073,Z 573.501,A -85,B 0,C 180,E1 -12188.793,E2 -12188.793} C_VEL
LIN {X 0,Y 376.932,Z 567.569,A -85,B 0,C 180,E1 -12190.736,E2 -12190.736} C_VEL
LIN {X 0,Y 378.25,Z 559.077,A -85,B 0,C 180,E1 -12193.064,E2 -12193.064} C_VEL
LIN {X 0,Y 379.725,Z 550.508,A -85,B 0,C 180,E1 -12195.033,E2 -12195.033} C_VEL
LIN {X 0,Y 381.699,Z 539.392,A -85,B 0,C 180,E1 -12197.164,E2 -12197.164} C_VEL
LIN {X 0,Y 383.783,Z 527.571,A -85,B 0,C 180,E1 -12199.058,E2 -12199.058} C_VEL
LIN {X 0,Y 385.748,Z 515.914,A -85,B 0,C 180,E1 -12200.642,E2 -12200.642} C_VEL
LIN {X 0,Y 387.734,Z 504.096,A -85,B 0,C 180,E1 -12202.017,E2 -12202.017} C_VEL
LIN {X 0,Y 389.98,Z 488.758,A -85,B 0,C 180,E1 -12203.508,E2 -12203.508} C_VEL
LIN {X 0,Y 391.966,Z 474.044,A -85,B 0,C 180,E1 -12204.667,E2 -12204.667} C_VEL
LIN {X 0,Y 393.715,Z 458.783,A -85,B 0,C 180,E1 -12205.646,E2 -12205.646} C_VEL
LIN {X 0,Y 395.244,Z 441.973,A -85,B 0,C 180,E1 -12206.49,E2 -12206.49} C_VEL
LIN {X 0,Y 396.464,Z 425.539,A -85,B 0,C 180,E1 -12207.088,E2 -12207.088} C_VEL
LIN {X 0,Y 397.275,Z 408.678,A -85,B 0,C 180,E1 -12207.5,E2 -12207.5} C_VEL
LIN {X 0,Y 401.829,Z 258.245,A -85,B 0,C 180,E1 -12210.389,E2 -12210.389} C_VEL
LIN {X 0,Y 393.054,Z 240.848,A -85,B 0,C 180,E1 -12211.753,E2 -12211.753} C_VEL
LIN {X 0,Y 385.396,Z 227.309,A -85,B 0,C 180,E1 -12212.988,E2 -12212.988} C_VEL
LIN {X 0,Y 377.429,Z 214.463,A -85,B 0,C 180,E1 -12214.332,E2 -12214.332} C_VEL
LIN {X 0,Y 376.495,Z 212.841,A -85,B 0,C 180,E1 -12214.518,E2 -12214.518} C_VEL
LIN {X 0,Y 375.958,Z 210.962,A -85,B 0,C 180,E1 -12214.98,E2 -12214.98} C_VEL
LIN {X 0,Y 375.948,Z 210.961,A -85,B 0,C 180,E1 -12218.045,E2 -12218.045} C_VEL
LIN {X 0,Y 375.996,Z 210.957,A -85,B 0,C 180,E1 -12221.473,E2 -12221.473} C_VEL
LIN {X 0,Y 376.051,Z 210.946,A -85,B 0,C 180,E1 -12224.832,E2 -12224.832} C_VEL
LIN {X 0,Y 376.042,Z 210.943,A -85,B 0,C 180,E1 -12228.136,E2 -12228.136} C_VEL
LIN {X 0,Y 376.193,Z 210.936,A -85,B 0,C 180,E1 -12231.94,E2 -12231.94} C_VEL
LIN {X 0,Y 376.159,Z 210.943,A -85,B 0,C 180,E1 -12234.64,E2 -12234.64} C_VEL
LIN {X 0,Y 376.345,Z 210.916,A -85,B 0,C 180,E1 -12237.86,E2 -12237.86} C_VEL
LIN {X 0,Y 376.482,Z 210.901,A -85,B 0,C 180,E1 -12240,E2 -12240} C_VEL
LIN {X 0,Y 376.178,Z 210.934,A -85,B 0,C 180,E1 -12243.213,E2 -12243.213} C_VEL
LIN {X 0,Y 376.235,Z 210.932,A -85,B 0,C 180,E1 -12246.435,E2 -12246.435} C_VEL
LIN {X 0,Y 376.113,Z 210.948,A -85,B 0,C 180,E1 -12249.682,E2 -12249.682} C_VEL
LIN {X 0,Y 376.083,Z 210.948,A -85,B 0,C 180,E1 -12253.658,E2 -12253.658} C_VEL
LIN {X 0,Y 376.037,Z 210.957,A -85,B 0,C 180,E1 -12257.607,E2 -12257.607} C_VEL
LIN {X 0,Y 375.972,Z 210.964,A -85,B 0,C 180,E1 -12260.832,E2 -12260.832} C_VEL
LIN {X 0,Y 375.988,Z 210.96,A -85,B 0,C 180,E1 -12264.282,E2 -12264.282} C_VEL
LIN {X 0,Y 376.014,Z 210.955,A -85,B 0,C 180,E1 -12266.652,E2 -12266.652} C_VEL
LIN {X 0,Y 375.959,Z 210.968,A -85,B 0,C 180,E1 -12270.313,E2 -12270.313} C_VEL
LIN {X 0,Y 375.954,Z 210.969,A -85,B 0,C 180,E1 -12274.112,E2 -12274.112} C_VEL
LIN {X 0,Y 375.948,Z 210.972,A -85,B 0,C 180,E1 -12276.742,E2 -12276.742} C_VEL
LIN {X 0,Y 375.984,Z 210.967,A -85,B 0,C 180,E1 -12279.971,E2 -12279.971} C_VEL
LIN {X 0,Y 375.925,Z 210.975,A -85,B 0,C 180,E1 -12283.766,E2 -12283.766} C_VEL
LIN {X 0,Y 375.93,Z 210.976,A -85,B 0,C 180,E1 -12286.811,E2 -12286.811} C_VEL
LIN {X 0,Y 375.952,Z 211.083,A -85,B 0,C 180,E1 -12288.652,E2 -12288.652} C_VEL
LIN {X 0,Y 381.115,Z 224.877,A -85,B 0,C 180,E1 -12291.602,E2 -12291.602} C_VEL
LIN {X 0,Y 382.425,Z 228.617,A -85,B 0,C 180,E1 -12292.314,E2 -12292.314} C_VEL
LIN {X 0,Y 391.278,Z 244.66,A -85,B 0,C 180,E1 -12293.773,E2 -12293.773} C_VEL
LIN {X 0,Y 400.349,Z 263.315,A -85,B 0,C 180,E1 -12295.208,E2 -12295.208} C_VEL
LIN {X 0,Y 401.583,Z 272.12,A -85,B 0,C 180,E1 -12295.537,E2 -12295.537} C_VEL
LIN {X 0,Y 396.498,Z 437.286,A -85,B 0,C 180,E1 -12298.726,E2 -12298.726} C_VEL
LIN {X 0,Y 395.184,Z 454.626,A -85,B 0,C 180,E1 -12299.251,E2 -12299.251} C_VEL
LIN {X 0,Y 393.723,Z 470.392,A -85,B 0,C 180,E1 -12299.94,E2 -12299.94} C_VEL
LIN {X 0,Y 392.065,Z 485.038,A -85,B 0,C 180,E1 -12300.761,E2 -12300.761} C_VEL
LIN {X 0,Y 390.149,Z 499.77,A -85,B 0,C 180,E1 -12301.781,E2 -12301.781} C_VEL
LIN {X 0,Y 387.938,Z 514.838,A -85,B 0,C 180,E1 -12303.07,E2 -12303.07} C_VEL
LIN {X 0,Y 385.757,Z 528.673,A -85,B 0,C 180,E1 -12304.507,E2 -12304.507} C_VEL
LIN {X 0,Y 383.756,Z 540.524,A -85,B 0,C 180,E1 -12305.954,E2 -12305.954} C_VEL
LIN {X 0,Y 381.894,Z 551.724,A -85,B 0,C 180,E1 -12307.552,E2 -12307.552} C_VEL
LIN {X 0,Y 380.028,Z 562.872,A -85,B 0,C 180,E1 -12309.429,E2 -12309.429} C_VEL
LIN {X 0,Y 378.215,Z 573.706,A -85,B 0,C 180,E1 -12311.586,E2 -12311.586} C_VEL
LIN {X 0,Y 377.08,Z 581.809,A -85,B 0,C 180,E1 -12313.488,E2 -12313.488} C_VEL
LIN {X 0,Y 375.913,Z 590.498,A -85,B 0,C 180,E1 -12315.934,E2 -12315.934} C_VEL
LIN {X 0,Y 375.115,Z 598.181,A -85,B 0,C 180,E1 -12318.655,E2 -12318.655} C_VEL
LIN {X 0,Y 374.673,Z 604.042,A -85,B 0,C 180,E1 -12321.37,E2 -12321.37} C_VEL
LIN {X 0,Y 374.552,Z 608.067,A -85,B 0,C 180,E1 -12323.973,E2 -12323.973} C_VEL
LIN {X 0,Y 374.477,Z 609.94,A -85,B 0,C 180,E1 -12325.695,E2 -12325.695} C_VEL
LIN {X 0,Y 374.47,Z 611.344,A -85,B 0,C 180,E1 -12327.849,E2 -12327.849} C_VEL
LIN {X 0,Y 374.55,Z 611.845,A -85,B 0,C 180,E1 -12330,E2 -12330} C_VEL
LIN {X 0,Y 374.471,Z 611.289,A -85,B 0,C 180,E1 -12332.151,E2 -12332.151} C_VEL
LIN {X 0,Y 374.477,Z 609.824,A -85,B 0,C 180,E1 -12334.305,E2 -12334.305} C_VEL
LIN {X 0,Y 374.559,Z 607.286,A -85,B 0,C 180,E1 -12336.464,E2 -12336.464} C_VEL
LIN {X 0,Y 374.674,Z 603.761,A -85,B 0,C 180,E1 -12338.631,E2 -12338.631} C_VEL
LIN {X 0,Y 374.96,Z 599.1,A -85,B 0,C 180,E1 -12340.803,E2 -12340.803} C_VEL
LIN {X 0,Y 375.579,Z 593.271,A -85,B 0,C 180,E1 -12342.977,E2 -12342.977} C_VEL
LIN {X 0,Y 376.312,Z 586.208,A -85,B 0,C 180,E1 -12345.157,E2 -12345.157} C_VEL
LIN {X 0,Y 377.683,Z 576.487,A -85,B 0,C 180,E1 -12347.601,E2 -12347.601} C_VEL
LIN {X 0,Y 379.177,Z 566.034,A -85,B 0,C 180,E1 -12349.771,E2 -12349.771} C_VEL
LIN {X 0,Y 380.881,Z 555.208,A -85,B 0,C 180,E1 -12351.656,E2 -12351.656} C_VEL
LIN {X 0,Y 382.682,Z 543.977,A -85,B 0,C 180,E1 -12353.328,E2 -12353.328} C_VEL
LIN {X 0,Y 384.641,Z 532.017,A -85,B 0,C 180,E1 -12354.85,E2 -12354.85} C_VEL
LIN {X 0,Y 386.653,Z 518.478,A -85,B 0,C 180,E1 -12356.299,E2 -12356.299} C_VEL
LIN {X 0,Y 388.594,Z 504.449,A -85,B 0,C 180,E1 -12357.555,E2 -12357.555} C_VEL
LIN {X 0,Y 390.512,Z 489.871,A -85,B 0,C 180,E1 -12358.631,E2 -12358.631} C_VEL
LIN {X 0,Y 392.329,Z 473.731,A -85,B 0,C 180,E1 -12359.587,E2 -12359.587} C_VEL
LIN {X 0,Y 393.746,Z 456.853,A -85,B 0,C 180,E1 -12360.355,E2 -12360.355} C_VEL
LIN {X 0,Y 394.953,Z 440.075,A -85,B 0,C 180,E1 -12360.881,E2 -12360.881} C_VEL
LIN {X 0,Y 395.765,Z 418.88,A -85,B 0,C 180,E1 -12361.319,E2 -12361.319} C_VEL
LIN {X 0,Y 399.831,Z 271.075,A -85,B 0,C 180,E1 -12364.115,E2 -12364.115} C_VEL
LIN {X 0,Y 398.17,Z 261.682,A -85,B 0,C 180,E1 -12364.472,E2 -12364.472} C_VEL
LIN {X 0,Y 386.32,Z 237.182,A -85,B 0,C 180,E1 -12366.169,E2 -12366.169} C_VEL
LIN {X 0,Y 382.262,Z 229.471,A -85,B 0,C 180,E1 -12366.784,E2 -12366.784} C_VEL
LIN {X 0,Y 377.729,Z 216.212,A -85,B 0,C 180,E1 -12369.242,E2 -12369.242} C_VEL
LIN {X 0,Y 375.939,Z 210.963,A -85,B 0,C 180,E1 -12370.265,E2 -12370.265} C_VEL
LIN {X 0,Y 375.927,Z 210.97,A -85,B 0,C 180,E1 -12373.766,E2 -12373.766} C_VEL
LIN {X 0,Y 375.931,Z 210.966,A -85,B 0,C 180,E1 -12376.811,E2 -12376.811} C_VEL
LIN {X 0,Y 375.941,Z 210.965,A -85,B 0,C 180,E1 -12380.535,E2 -12380.535} C_VEL
LIN {X 0,Y 375.961,Z 210.952,A -85,B 0,C 180,E1 -12383.496,E2 -12383.496} C_VEL
LIN {X 0,Y 375.958,Z 210.966,A -85,B 0,C 180,E1 -12385.888,E2 -12385.888} C_VEL
LIN {X 0,Y 375.962,Z 210.961,A -85,B 0,C 180,E1 -12389.687,E2 -12389.687} C_VEL
LIN {X 0,Y 376.017,Z 210.942,A -85,B 0,C 180,E1 -12393.348,E2 -12393.348} C_VEL
LIN {X 0,Y 375.994,Z 210.966,A -85,B 0,C 180,E1 -12396.888,E2 -12396.888} C_VEL
LIN {X 0,Y 375.993,Z 210.939,A -85,B 0,C 180,E1 -12400.339,E2 -12400.339} C_VEL
LIN {X 0,Y 376.023,Z 210.956,A -85,B 0,C 180,E1 -12403.719,E2 -12403.719} C_VEL
LIN {X 0,Y 376.101,Z 210.928,A -85,B 0,C 180,E1 -12407.042,E2 -12407.042} C_VEL
LIN {X 0,Y 376.111,Z 210.933,A -85,B 0,C 180,E1 -12410.318,E2 -12410.318} C_VEL
LIN {X 0,Y 376.226,Z 210.93,A -85,B 0,C 180,E1 -12413.565,E2 -12413.565} C_VEL
LIN {X 0,Y 376.348,Z 210.884,A -85,B 0,C 180,E1 -12417.86,E2 -12417.86} C_VEL
LIN {X 0,Y 376.484,Z 210.892,A -85,B 0,C 180,E1 -12420,E2 -12420} C_VEL
LIN {X 0,Y 376.181,Z 210.933,A -85,B 0,C 180,E1 -12423.213,E2 -12423.213} C_VEL
LIN {X 0,Y 376.222,Z 210.923,A -85,B 0,C 180,E1 -12426.632,E2 -12426.632} C_VEL
LIN {X 0,Y 376.116,Z 210.945,A -85,B 0,C 180,E1 -12429.681,E2 -12429.681} C_VEL
LIN {X 0,Y 376.087,Z 210.94,A -85,B 0,C 180,E1 -12433.658,E2 -12433.658} C_VEL
LIN {X 0,Y 376.041,Z 210.944,A -85,B 0,C 180,E1 -12437.607,E2 -12437.607} C_VEL
LIN {X 0,Y 375.976,Z 210.959,A -85,B 0,C 180,E1 -12440.832,E2 -12440.832} C_VEL
LIN {X 0,Y 375.992,Z 210.949,A -85,B 0,C 180,E1 -12444.282,E2 -12444.282} C_VEL
LIN {X 0,Y 376.018,Z 210.95,A -85,B 0,C 180,E1 -12446.652,E2 -12446.652} C_VEL
LIN {X 0,Y 375.975,Z 210.963,A -85,B 0,C 180,E1 -12449.079,E2 -12449.079} C_VEL
LIN {X 0,Y 375.949,Z 210.954,A -85,B 0,C 180,E1 -12452.828,E2 -12452.828} C_VEL
LIN {X 0,Y 375.956,Z 210.968,A -85,B 0,C 180,E1 -12455.415,E2 -12455.415} C_VEL
LIN {X 0,Y 375.974,Z 210.949,A -85,B 0,C 180,E1 -12458.271,E2 -12458.271} C_VEL
LIN {X 0,Y 375.933,Z 210.97,A -85,B 0,C 180,E1 -12461.601,E2 -12461.601} C_VEL
LIN {X 0,Y 375.925,Z 210.965,A -85,B 0,C 180,E1 -12465.269,E2 -12465.269} C_VEL
LIN {X 0,Y 375.932,Z 210.96,A -85,B 0,C 180,E1 -12468.399,E2 -12468.399} C_VEL
LIN {X 0,Y 375.971,Z 210.965,A -85,B 0,C 180,E1 -12471.73,E2 -12471.73} C_VEL
LIN {X 0,Y 375.979,Z 210.96,A -85,B 0,C 180,E1 -12475.333,E2 -12475.333} C_VEL
LIN {X 0,Y 375.956,Z 210.956,A -85,B 0,C 180,E1 -12478.438,E2 -12478.438} C_VEL
LIN {X 0,Y 375.982,Z 210.957,A -85,B 0,C 180,E1 -12482.14,E2 -12482.14} C_VEL
LIN {X 0,Y 376.006,Z 210.96,A -85,B 0,C 180,E1 -12484.539,E2 -12484.539} C_VEL
LIN {X 0,Y 375.968,Z 210.966,A -85,B 0,C 180,E1 -12488.046,E2 -12488.046} C_VEL
LIN {X 0,Y 376.008,Z 210.934,A -85,B 0,C 180,E1 -12491.473,E2 -12491.473} C_VEL
LIN {X 0,Y 376.058,Z 210.943,A -85,B 0,C 180,E1 -12494.832,E2 -12494.832} C_VEL
LIN {X 0,Y 376.051,Z 210.957,A -85,B 0,C 180,E1 -12498.136,E2 -12498.136} C_VEL
LIN {X 0,Y 376.104,Z 211.133,A -85,B 0,C 180,E1 -12498.569,E2 -12498.569} C_VEL
LIN {X 0,Y 376.661,Z 213.018,A -85,B 0,C 180,E1 -12498.738,E2 -12498.738} C_VEL
LIN {X 0,Y 378.673,Z 216.219,A -85,B 0,C 180,E1 -12499.032,E2 -12499.032} C_VEL
LIN {X 0,Y 385.979,Z 229.085,A -85,B 0,C 180,E1 -12500.098,E2 -12500.098} C_VEL
LIN {X 0,Y 394.027,Z 244.595,A -85,B 0,C 180,E1 -12501.248,E2 -12501.248} C_VEL
LIN {X 0,Y 400.062,Z 257.555,A -85,B 0,C 180,E1 -12502.099,E2 -12502.099} C_VEL
LIN {X 0,Y 395.459,Z 417.553,A -85,B 0,C 180,E1 -12505.141,E2 -12505.141} C_VEL
LIN {X 0,Y 394.492,Z 433.944,A -85,B 0,C 180,E1 -12505.648,E2 -12505.648} C_VEL
LIN {X 0,Y 393.16,Z 450.169,A -85,B 0,C 180,E1 -12506.349,E2 -12506.349} C_VEL
LIN {X 0,Y 391.775,Z 464.768,A -85,B 0,C 180,E1 -12507.172,E2 -12507.172} C_VEL
LIN {X 0,Y 390.103,Z 479.424,A -85,B 0,C 180,E1 -12508.193,E2 -12508.193} C_VEL
LIN {X 0,Y 388.1,Z 494.432,A -85,B 0,C 180,E1 -12509.481,E2 -12509.481} C_VEL
LIN {X 0,Y 386.02,Z 508.291,A -85,B 0,C 180,E1 -12510.916,E2 -12510.916} C_VEL
LIN {X 0,Y 384.373,Z 519.339,A -85,B 0,C 180,E1 -12512.266,E2 -12512.266} C_VEL
LIN {X 0,Y 383.076,Z 523.788,A -85,B 0,C 180,E1 -12512.826,E2 -12512.826} C_VEL
LIN {X 0,Y 376.005,Z 536.247,A -85,B 0,C 180,E1 -12514.428,E2 -12514.428} C_VEL
LIN {X 0,Y 374.312,Z 540.185,A -85,B 0,C 180,E1 -12515.049,E2 -12515.049} C_VEL
LIN {X 0,Y 373.998,Z 541.43,A -85,B 0,C 180,E1 -12515.274,E2 -12515.274} C_VEL
LIN {X 0,Y 372.274,Z 551.701,A -85,B 0,C 180,E1 -12517.321,E2 -12517.321} C_VEL
LIN {X 0,Y 370.979,Z 559.614,A -85,B 0,C 180,E1 -12519.176,E2 -12519.176} C_VEL
LIN {X 0,Y 369.691,Z 567.961,A -85,B 0,C 180,E1 -12521.514,E2 -12521.514} C_VEL
LIN {X 0,Y 368.832,Z 574.25,A -85,B 0,C 180,E1 -12523.642,E2 -12523.642} C_VEL
LIN {X 0,Y 368.136,Z 580.059,A -85,B 0,C 180,E1 -12526.07,E2 -12526.07} C_VEL
LIN {X 0,Y 367.773,Z 583.325,A -85,B 0,C 180,E1 -12527.803,E2 -12527.803} C_VEL
LIN {X 0,Y 367.385,Z 587.067,A -85,B 0,C 180,E1 -12530.388,E2 -12530.388} C_VEL
LIN {X 0,Y 367.143,Z 589.571,A -85,B 0,C 180,E1 -12533.244,E2 -12533.244} C_VEL
LIN {X 0,Y 367.116,Z 590.408,A -85,B 0,C 180,E1 -12535.874,E2 -12535.874} C_VEL
LIN {X 0,Y 367.21,Z 589.973,A -85,B 0,C 180,E1 -12538.311,E2 -12538.311} C_VEL
LIN {X 0,Y 367.316,Z 588.588,A -85,B 0,C 180,E1 -12540.571,E2 -12540.571} C_VEL
LIN {X 0,Y 367.549,Z 586.229,A -85,B 0,C 180,E1 -12542.719,E2 -12542.719} C_VEL
LIN {X 0,Y 368.008,Z 582.845,A -85,B 0,C 180,E1 -12544.953,E2 -12544.953} C_VEL
LIN {X 0,Y 368.627,Z 577.408,A -85,B 0,C 180,E1 -12547.595,E2 -12547.595} C_VEL
LIN {X 0,Y 369.343,Z 572.145,A -85,B 0,C 180,E1 -12549.601,E2 -12549.601} C_VEL
LIN {X 0,Y 370.517,Z 564.662,A -85,B 0,C 180,E1 -12551.969,E2 -12551.969} C_VEL
LIN {X 0,Y 371.96,Z 556.463,A -85,B 0,C 180,E1 -12554.111,E2 -12554.111} C_VEL
LIN {X 0,Y 373.541,Z 547.483,A -85,B 0,C 180,E1 -12556.078,E2 -12556.078} C_VEL
LIN {X 0,Y 375.678,Z 536.182,A -85,B 0,C 180,E1 -12558.167,E2 -12558.167} C_VEL
LIN {X 0,Y 377.984,Z 523.79,A -85,B 0,C 180,E1 -12560.082,E2 -12560.082} C_VEL
LIN {X 0,Y 380.244,Z 510.818,A -85,B 0,C 180,E1 -12561.768,E2 -12561.768} C_VEL
LIN {X 0,Y 382.556,Z 496.977,A -85,B 0,C 180,E1 -12563.268,E2 -12563.268} C_VEL
LIN {X 0,Y 384.685,Z 482.599,A -85,B 0,C 180,E1 -12564.554,E2 -12564.554} C_VEL
LIN {X 0,Y 386.631,Z 467.904,A -85,B 0,C 180,E1 -12565.633,E2 -12565.633} C_VEL
LIN {X 0,Y 388.318,Z 452.35,A -85,B 0,C 180,E1 -12566.555,E2 -12566.555} C_VEL
LIN {X 0,Y 389.715,Z 437.23,A -85,B 0,C 180,E1 -12567.248,E2 -12567.248} C_VEL
LIN {X 0,Y 390.817,Z 420.434,A -85,B 0,C 180,E1 -12567.799,E2 -12567.799} C_VEL
LIN {X 0,Y 391.799,Z 392.962,A -85,B 0,C 180,E1 -12568.374,E2 -12568.374} C_VEL
LIN {X 0,Y 396.11,Z 260.691,A -85,B 0,C 180,E1 -12570.947,E2 -12570.947} C_VEL
LIN {X 0,Y 388.01,Z 244.597,A -85,B 0,C 180,E1 -12572.248,E2 -12572.248} C_VEL
LIN {X 0,Y 380.05,Z 230.434,A -85,B 0,C 180,E1 -12573.579,E2 -12573.579} C_VEL
LIN {X 0,Y 371.636,Z 216.943,A -85,B 0,C 180,E1 -12575.055,E2 -12575.055} C_VEL
LIN {X 0,Y 369.319,Z 213.547,A -85,B 0,C 180,E1 -12575.474,E2 -12575.474} C_VEL
LIN {X 0,Y 368.915,Z 211.84,A -85,B 0,C 180,E1 -12575.838,E2 -12575.838} C_VEL
LIN {X 0,Y 368.913,Z 211.845,A -85,B 0,C 180,E1 -12578.981,E2 -12578.981} C_VEL
LIN {X 0,Y 368.985,Z 211.837,A -85,B 0,C 180,E1 -12582.257,E2 -12582.257} C_VEL
LIN {X 0,Y 369.031,Z 211.832,A -85,B 0,C 180,E1 -12586.228,E2 -12586.228} C_VEL
LIN {X 0,Y 369.057,Z 211.827,A -85,B 0,C 180,E1 -12590.131,E2 -12590.131} C_VEL
LIN {X 0,Y 369.18,Z 211.807,A -85,B 0,C 180,E1 -12593.441,E2 -12593.441} C_VEL
LIN {X 0,Y 369.31,Z 211.793,A -85,B 0,C 180,E1 -12597.819,E2 -12597.819} C_VEL
LIN {X 0,Y 369.452,Z 211.777,A -85,B 0,C 180,E1 -12600,E2 -12600} C_VEL
LIN {X 0,Y 369.31,Z 211.796,A -85,B 0,C 180,E1 -12602.181,E2 -12602.181} C_VEL
LIN {X 0,Y 369.195,Z 211.81,A -85,B 0,C 180,E1 -12606.558,E2 -12606.558} C_VEL
LIN {X 0,Y 369.061,Z 211.828,A -85,B 0,C 180,E1 -12609.868,E2 -12609.868} C_VEL
LIN {X 0,Y 369.031,Z 211.826,A -85,B 0,C 180,E1 -12613.772,E2 -12613.772} C_VEL
LIN {X 0,Y 368.995,Z 211.836,A -85,B 0,C 180,E1 -12617.769,E2 -12617.769} C_VEL
LIN {X 0,Y 368.923,Z 211.842,A -85,B 0,C 180,E1 -12621.22,E2 -12621.22} C_VEL
LIN {X 0,Y 368.952,Z 211.837,A -85,B 0,C 180,E1 -12624.776,E2 -12624.776} C_VEL
LIN {X 0,Y 368.957,Z 211.836,A -85,B 0,C 180,E1 -12627.204,E2 -12627.204} C_VEL
LIN {X 0,Y 368.924,Z 211.844,A -85,B 0,C 180,E1 -12630.954,E2 -12630.954} C_VEL
LIN {X 0,Y 368.923,Z 211.848,A -85,B 0,C 180,E1 -12635.002,E2 -12635.002} C_VEL
LIN {X 0,Y 368.904,Z 211.85,A -85,B 0,C 180,E1 -12638.641,E2 -12638.641} C_VEL
LIN {X 0,Y 368.876,Z 211.853,A -85,B 0,C 180,E1 -12642.01,E2 -12642.01} C_VEL
LIN {X 0,Y 368.875,Z 211.855,A -85,B 0,C 180,E1 -12645.176,E2 -12645.176} C_VEL
LIN {X 0,Y 368.902,Z 211.921,A -85,B 0,C 180,E1 -12647.765,E2 -12647.765} C_VEL
LIN {X 0,Y 374.246,Z 226.042,A -85,B 0,C 180,E1 -12650.915,E2 -12650.915} C_VEL
LIN {X 0,Y 375.106,Z 228.328,A -85,B 0,C 180,E1 -12651.36,E2 -12651.36} C_VEL
LIN {X 0,Y 385.379,Z 246.669,A -85,B 0,C 180,E1 -12653.126,E2 -12653.126} C_VEL
LIN {X 0,Y 394.858,Z 266.216,A -85,B 0,C 180,E1 -12654.682,E2 -12654.682} C_VEL
LIN {X 0,Y 395.814,Z 272.593,A -85,B 0,C 180,E1 -12654.935,E2 -12654.935} C_VEL
LIN {X 0,Y 391.555,Z 405.04,A -85,B 0,C 180,E1 -12657.508,E2 -12657.508} C_VEL
LIN {X 0,Y 390.456,Z 438.21,A -85,B 0,C 180,E1 -12658.193,E2 -12658.193} C_VEL
LIN {X 0,Y 389.132,Z 455.117,A -85,B 0,C 180,E1 -12658.719,E2 -12658.719} C_VEL
LIN {X 0,Y 387.608,Z 470.685,A -85,B 0,C 180,E1 -12659.415,E2 -12659.415} C_VEL
LIN {X 0,Y 385.882,Z 485.205,A -85,B 0,C 180,E1 -12660.245,E2 -12660.245} C_VEL
LIN {X 0,Y 383.896,Z 499.837,A -85,B 0,C 180,E1 -12661.279,E2 -12661.279} C_VEL
LIN {X 0,Y 381.594,Z 514.849,A -85,B 0,C 180,E1 -12662.585,E2 -12662.585} C_VEL
LIN {X 0,Y 379.26,Z 528.633,A -85,B 0,C 180,E1 -12664.038,E2 -12664.038} C_VEL
LIN {X 0,Y 377.219,Z 540.455,A -85,B 0,C 180,E1 -12665.51,E2 -12665.51} C_VEL
LIN {X 0,Y 375.271,Z 551.645,A -85,B 0,C 180,E1 -12667.133,E2 -12667.133} C_VEL
LIN {X 0,Y 373.285,Z 562.772,A -85,B 0,C 180,E1 -12669.04,E2 -12669.04} C_VEL
LIN {X 0,Y 371.523,Z 572.77,A -85,B 0,C 180,E1 -12671.055,E2 -12671.055} C_VEL
LIN {X 0,Y 370.2,Z 581.661,A -85,B 0,C 180,E1 -12673.172,E2 -12673.172} C_VEL
LIN {X 0,Y 368.928,Z 590.335,A -85,B 0,C 180,E1 -12675.662,E2 -12675.662} C_VEL
LIN {X 0,Y 368.072,Z 598.009,A -85,B 0,C 180,E1 -12678.435,E2 -12678.435} C_VEL
LIN {X 0,Y 367.587,Z 603.863,A -85,B 0,C 180,E1 -12681.202,E2 -12681.202} C_VEL
LIN {X 0,Y 367.467,Z 608.077,A -85,B 0,C 180,E1 -12684.001,E2 -12684.001} C_VEL
LIN {X 0,Y 367.385,Z 609.747,A -85,B 0,C 180,E1 -12685.612,E2 -12685.612} C_VEL
LIN {X 0,Y 367.368,Z 611.145,A -85,B 0,C 180,E1 -12687.808,E2 -12687.808} C_VEL
LIN {X 0,Y 367.453,Z 611.636,A -85,B 0,C 180,E1 -12690,E2 -12690} C_VEL
LIN {X 0,Y 367.369,Z 611.075,A -85,B 0,C 180,E1 -12692.193,E2 -12692.193} C_VEL
LIN {X 0,Y 367.386,Z 609.599,A -85,B 0,C 180,E1 -12694.389,E2 -12694.389} C_VEL
LIN {X 0,Y 367.476,Z 607.054,A -85,B 0,C 180,E1 -12696.589,E2 -12696.589} C_VEL
LIN {X 0,Y 367.589,Z 603.512,A -85,B 0,C 180,E1 -12698.798,E2 -12698.798} C_VEL
LIN {X 0,Y 367.929,Z 598.842,A -85,B 0,C 180,E1 -12701.012,E2 -12701.012} C_VEL
LIN {X 0,Y 368.556,Z 592.996,A -85,B 0,C 180,E1 -12703.228,E2 -12703.228} C_VEL
LIN {X 0,Y 369.518,Z 584.892,A -85,B 0,C 180,E1 -12705.725,E2 -12705.725} C_VEL
LIN {X 0,Y 370.798,Z 576.172,A -85,B 0,C 180,E1 -12707.939,E2 -12707.939} C_VEL
LIN {X 0,Y 372.382,Z 565.704,A -85,B 0,C 180,E1 -12710.147,E2 -12710.147} C_VEL
LIN {X 0,Y 374.175,Z 554.851,A -85,B 0,C 180,E1 -12712.065,E2 -12712.065} C_VEL
LIN {X 0,Y 376.103,Z 543.318,A -85,B 0,C 180,E1 -12713.801,E2 -12713.801} C_VEL
LIN {X 0,Y 378.251,Z 530.426,A -85,B 0,C 180,E1 -12715.447,E2 -12715.447} C_VEL
LIN {X 0,Y 380.391,Z 516.708,A -85,B 0,C 180,E1 -12716.914,E2 -12716.914} C_VEL
LIN {X 0,Y 382.552,Z 501.874,A -85,B 0,C 180,E1 -12718.219,E2 -12718.219} C_VEL
LIN {X 0,Y 384.507,Z 487.237,A -85,B 0,C 180,E1 -12719.271,E2 -12719.271} C_VEL
LIN {X 0,Y 386.226,Z 471.634,A -85,B 0,C 180,E1 -12720.177,E2 -12720.177} C_VEL
LIN {X 0,Y 387.578,Z 455.902,A -85,B 0,C 180,E1 -12720.89,E2 -12720.89} C_VEL
LIN {X 0,Y 388.849,Z 438.82,A -85,B 0,C 180,E1 -12721.421,E2 -12721.421} C_VEL
LIN {X 0,Y 389.691,Z 415.697,A -85,B 0,C 180,E1 -12721.893,E2 -12721.893} C_VEL
LIN {X 0,Y 393.832,Z 272.093,A -85,B 0,C 180,E1 -12724.649,E2 -12724.649} C_VEL
LIN {X 0,Y 392.44,Z 264.574,A -85,B 0,C 180,E1 -12724.947,E2 -12724.947} C_VEL
LIN {X 0,Y 381.48,Z 241.617,A -85,B 0,C 180,E1 -12726.564,E2 -12726.564} C_VEL
LIN {X 0,Y 374.953,Z 229.339,A -85,B 0,C 180,E1 -12727.555,E2 -12727.555} C_VEL
LIN {X 0,Y 370.819,Z 217.247,A -85,B 0,C 180,E1 -12729.864,E2 -12729.864} C_VEL
LIN {X 0,Y 368.894,Z 211.846,A -85,B 0,C 180,E1 -12730.948,E2 -12730.948} C_VEL
LIN {X 0,Y 368.88,Z 211.845,A -85,B 0,C 180,E1 -12733.616,E2 -12733.616} C_VEL
LIN {X 0,Y 368.883,Z 211.842,A -85,B 0,C 180,E1 -12736.696,E2 -12736.696} C_VEL
LIN {X 0,Y 368.905,Z 211.835,A -85,B 0,C 180,E1 -12739.644,E2 -12739.644} C_VEL
LIN {X 0,Y 368.897,Z 211.833,A -85,B 0,C 180,E1 -12743.145,E2 -12743.145} C_VEL
LIN {X 0,Y 368.894,Z 211.847,A -85,B 0,C 180,E1 -12746.462,E2 -12746.462} C_VEL
LIN {X 0,Y 368.927,Z 211.828,A -85,B 0,C 180,E1 -12749.046,E2 -12749.046} C_VEL
LIN {X 0,Y 368.961,Z 211.826,A -85,B 0,C 180,E1 -12752.797,E2 -12752.797} C_VEL
LIN {X 0,Y 368.943,Z 211.836,A -85,B 0,C 180,E1 -12756.113,E2 -12756.113} C_VEL
LIN {X 0,Y 368.933,Z 211.821,A -85,B 0,C 180,E1 -12759.947,E2 -12759.947} C_VEL
LIN {X 0,Y 368.966,Z 211.835,A -85,B 0,C 180,E1 -12763.398,E2 -12763.398} C_VEL
LIN {X 0,Y 369.055,Z 211.807,A -85,B 0,C 180,E1 -12766.79,E2 -12766.79} C_VEL
LIN {X 0,Y 369.061,Z 211.808,A -85,B 0,C 180,E1 -12770.132,E2 -12770.132} C_VEL
LIN {X 0,Y 369.184,Z 211.807,A -85,B 0,C 180,E1 -12773.441,E2 -12773.441} C_VEL
LIN {X 0,Y 369.313,Z 211.759,A -85,B 0,C 180,E1 -12777.819,E2 -12777.819} C_VEL
LIN {X 0,Y 369.454,Z 211.768,A -85,B 0,C 180,E1 -12780,E2 -12780} C_VEL
LIN {X 0,Y 369.313,Z 211.796,A -85,B 0,C 180,E1 -12782.181,E2 -12782.181} C_VEL
LIN {X 0,Y 369.193,Z 211.8,A -85,B 0,C 180,E1 -12786.617,E2 -12786.617} C_VEL
LIN {X 0,Y 369.065,Z 211.821,A -85,B 0,C 180,E1 -12789.868,E2 -12789.868} C_VEL
LIN {X 0,Y 369.035,Z 211.82,A -85,B 0,C 180,E1 -12793.772,E2 -12793.772} C_VEL
LIN {X 0,Y 368.999,Z 211.818,A -85,B 0,C 180,E1 -12797.768,E2 -12797.768} C_VEL
LIN {X 0,Y 368.927,Z 211.837,A -85,B 0,C 180,E1 -12801.22,E2 -12801.22} C_VEL
LIN {X 0,Y 368.955,Z 211.823,A -85,B 0,C 180,E1 -12804.775,E2 -12804.775} C_VEL
LIN {X 0,Y 368.985,Z 211.834,A -85,B 0,C 180,E1 -12808.436,E2 -12808.436} C_VEL
LIN {X 0,Y 368.898,Z 211.83,A -85,B 0,C 180,E1 -12812.238,E2 -12812.238} C_VEL
LIN {X 0,Y 368.927,Z 211.841,A -85,B 0,C 180,E1 -12815.002,E2 -12815.002} C_VEL
LIN {X 0,Y 368.908,Z 211.831,A -85,B 0,C 180,E1 -12818.641,E2 -12818.641} C_VEL
LIN {X 0,Y 368.88,Z 211.844,A -85,B 0,C 180,E1 -12822.009,E2 -12822.009} C_VEL
LIN {X 0,Y 368.878,Z 211.841,A -85,B 0,C 180,E1 -12825.176,E2 -12825.176} C_VEL
LIN {X 0,Y 368.881,Z 211.839,A -85,B 0,C 180,E1 -12828.178,E2 -12828.178} C_VEL
LIN {X 0,Y 368.906,Z 211.847,A -85,B 0,C 180,E1 -12831.36,E2 -12831.36} C_VEL
LIN {X 0,Y 368.935,Z 211.834,A -85,B 0,C 180,E1 -12835.146,E2 -12835.146} C_VEL
LIN {X 0,Y 368.928,Z 211.832,A -85,B 0,C 180,E1 -12839.046,E2 -12839.046} C_VEL
LIN {X 0,Y 368.975,Z 211.833,A -85,B 0,C 180,E1 -12841.564,E2 -12841.564} C_VEL
LIN {X 0,Y 368.999,Z 211.833,A -85,B 0,C 180,E1 -12844.02,E2 -12844.02} C_VEL
LIN {X 0,Y 368.935,Z 211.844,A -85,B 0,C 180,E1 -12847.605,E2 -12847.605} C_VEL
LIN {X 0,Y 368.957,Z 211.809,A -85,B 0,C 180,E1 -12851.106,E2 -12851.106} C_VEL
LIN {X 0,Y 368.998,Z 211.827,A -85,B 0,C 180,E1 -12854.535,E2 -12854.535} C_VEL
LIN {X 0,Y 369.032,Z 211.825,A -85,B 0,C 180,E1 -12857.838,E2 -12857.838} C_VEL
LIN {X 0,Y 369.998,Z 214.665,A -85,B 0,C 180,E1 -12858.034,E2 -12858.034} C_VEL
LIN {X 0,Y 371.585,Z 216.95,A -85,B 0,C 180,E1 -12858.27,E2 -12858.27} C_VEL
LIN {X 0,Y 378.702,Z 229.096,A -85,B 0,C 180,E1 -12859.339,E2 -12859.339} C_VEL
LIN {X 0,Y 386.575,Z 243.936,A -85,B 0,C 180,E1 -12860.499,E2 -12860.499} C_VEL
LIN {X 0,Y 394.029,Z 259.676,A -85,B 0,C 180,E1 -12861.582,E2 -12861.582} C_VEL
LIN {X 0,Y 389.308,Z 417.538,A -85,B 0,C 180,E1 -12864.626,E2 -12864.626} C_VEL
LIN {X 0,Y 388.25,Z 434.631,A -85,B 0,C 180,E1 -12865.161,E2 -12865.161} C_VEL
LIN {X 0,Y 386.948,Z 449.939,A -85,B 0,C 180,E1 -12865.834,E2 -12865.834} C_VEL
LIN {X 0,Y 385.406,Z 465.618,A -85,B 0,C 180,E1 -12866.733,E2 -12866.733} C_VEL
LIN {X 0,Y 383.655,Z 480.198,A -85,B 0,C 180,E1 -12867.769,E2 -12867.769} C_VEL
LIN {X 0,Y 381.803,Z 493.714,A -85,B 0,C 180,E1 -12868.945,E2 -12868.945} C_VEL
LIN {X 0,Y 379.692,Z 507.306,A -85,B 0,C 180,E1 -12870.35,E2 -12870.35} C_VEL
LIN {X 0,Y 377.662,Z 520.183,A -85,B 0,C 180,E1 -12871.94,E2 -12871.94} C_VEL
LIN {X 0,Y 375.516,Z 532.614,A -85,B 0,C 180,E1 -12873.755,E2 -12873.755} C_VEL
LIN {X 0,Y 373.998,Z 541.43,A -85,B 0,C 180,E1 -12875.274,E2 -12875.274} C_VEL
LIN {X 0,Y 372.689,Z 545.234,A -85,B 0,C 180,E1 -12875.945,E2 -12875.945} C_VEL
LIN {X 0,Y 365.85,Z 555.758,A -85,B 0,C 180,E1 -12877.918,E2 -12877.918} C_VEL
LIN {X 0,Y 364.32,Z 558.961,A -85,B 0,C 180,E1 -12878.658,E2 -12878.658} C_VEL
LIN {X 0,Y 364.07,Z 559.988,A -85,B 0,C 180,E1 -12878.919,E2 -12878.919} C_VEL
